// TwinCAT 3 PLC project Untitled1
// ProgramVersion: 3.1.4024.0
// libraries:
//   CmpBitmapPool, * (System)
//   Tc2_EtherCAT, * (Beckhoff Automation GmbH)
//   Tc2_MC2, * (Beckhoff Automation GmbH)
//   Tc2_ModbusSrv, * (Beckhoff Automation GmbH)
//   Tc2_Standard, * (Beckhoff Automation GmbH)
//   Tc2_SUPS, * (Beckhoff Automation GmbH)
//   Tc2_System, * (Beckhoff Automation GmbH)
//   Tc2_Utilities, * (Beckhoff Automation GmbH)
//   Tc3_Module, * (Beckhoff Automation GmbH)
//   Tc3_PackML_V2, * (Beckhoff Automation GmbH)
//   Util, * (System)
//   VisuDialogs, * (System)
// project tree:
//   02DUTs/ E_PMLUserUnitMode.TcDUT, E_UnitName.TcDUT, ST_ChangeIntoProduction.TcDUT (not stored), ST_UnitInfo.TcDUT (not stored)
//   Ads/ BarcodeVerificationResult.TcDUT (not stored), CurrentAirPressureState.TcDUT, DigitalInputStatus.TcDUT (not stored), DigitalOutputStatus.TcDUT (not stored), EStopStatus.TcDUT (not stored), E_SAFETYDOOR.TcDUT, E_SafetyStates.TcDUT (not stored), FB_AirPressure_Subsystem.TcPOU, FB_Application.TcPOU, FB_Light_tower_module.TcPOU (not stored), FB_Safety_module.TcPOU, FB_Tote_Subsystem.TcPOU, MachineControlCommand.TcDUT (not stored), MachineStatus.TcDUT (not stored), SafetyDoorStatus.TcDUT (not stored), SafetyStatus.TcDUT (not stored), StationMode.TcDUT (not stored), ST_LightTower.TcDUT (not stored)
//   GVLs/ GVL.TcGVL, GVL_IOLink.TcGVL (not stored), G_HMI.TcGVL, G_IO.TcGVL, ST_IO_16.TcDUT (not stored), ST_SafetyIO.TcDUT (not stored)
//   / EtherCAT_Task.TcTTO (not stored), GlobalTextList.TcGTLO, MianTask.TcTTO (not stored), VisualizationManager.TcVMO (not stored), VISU_TASK.TcTTO (not stored)
//   Mian/axis/ AxisHMI_Ex.TcVIS (not stored), E_HomingSteps.TcDUT (not stored), FB_MotionAxis_MC.TcPOU (not stored), MC_HomeAxis.TcPOU (not stored), ST_MotionAxis_MC.TcDUT
//   Mian/DUTs/ Buffer_roller.TcDUT (not stored), E_Condition.TcDUT (not stored), E_LoadingStates.TcDUT, E_SampleStates.TcDUT (not stored), E_RollerStates.TcDUT (not stored), E_topic_sample.TcDUT (not stored), E_Transfer.TcDUT (not stored), E_WorkingStates.TcDUT, FB_DigitalInput.TcPOU (not stored), FB_GPWM.TcPOU (not stored), Roller.TcDUT (not stored), ServerityLevelType.TcDUT (not stored), ST_control_pannel.TcDUT (not stored), ST_EVENT.TcDUT (not stored), ST_safetyDoor.TcDUT (not stored), ToteStatus.TcDUT, Valve.TcDUT (not stored)
//   Mian/ FB_mcp.TcPOU (not stored), FB_Generic.TcPOU, FB_Machine.TcPOU, FB_Sample.TcPOU, FB_Visu.TcPOU, I_Common.TcIO, MAIN.TcPOU
//   Mian/statemachine/ Prepare_Date_Time.TcPOU (not stored)
//   PubSub/ E_Topics.TcDUT, I_PubSubService.TcIO, I_SubCallback.TcIO (not stored), KeyAndValue.TcDUT (not stored), PubSubData.TcDUT (not stored), PubSubService.TcPOU, SubscriberCell.TcDUT
//   VISUs/ ImagePool.TcIPO (not stored), visu_main.TcVIS
//   VISUs/Templates/ VIS_TemplateCommand.TcVIS, VIS_TemplateKeys.TcVIS, VIS_TemplateMachine.TcVIS, VIS_TemplatePMLStateModel.TcVIS (not stored), VIS_TemplateToProduction.TcVIS (not stored)
//   VISUs/VISUs/ Menu.TcVIS, visu_sample.TcVIS (not stored), visu_manual.TcVIS, visu_operation.TcVIS, v_alarm.TcVIS
// real-time tasks:
//   TASK PlcTask: cycle T#4ms, priority 20, ADS port 350
//   TASK EtherCAT_Task: cycle T#2ms, priority 2, ADS port 351
//   TASK VISU_TASK: cycle T#100000us, priority 30, ADS port 352
// motion (NC):
//   TASK NC-Task 1 SAF: cycle T#2ms, priority 4, ADS port 501
//   TASK NC-Task 1 SVB: cycle T#10ms, priority 8, ADS port 511
//   AXIS buffer_stopper (id 1)
//     PositionAreaControl: Enable=false
//     OtherSettings: AllowMotionCmdToSlave=true
//     encoder EncType=19
//       EncPara: ScaleFactorNumerator=36, ScaleFactorDenominator=8388608, MaxCount=#xffffffff, ReferenceSystem=1
//         Inc: RefSoftSyncMask=#x00800000
//     drive DrvType=16
//       DrvPara: MaxCount=#xffffffff, DriveControlDWord=#x00000100
//         Analog: TorqueSetpointScale=10, ScaleFactorActTorque=0.1
//         TimeComp: TaskDelayCycles=1
//     controller CtrType=1
//       CtrPara: PriorControlFactor=1
//         PosDiffControl: Enable=false
//         Observer: BandWidth=20
//   AXIS lift_motor (id 3)
//     PositionAreaControl: Enable=false
//     OtherSettings: AllowMotionCmdToSlave=true
//     encoder EncType=19
//       EncPara: ScaleFactorNumerator=3.97364299e-07, MaxCount=#xffffffff, ReferenceSystem=1
//     drive DrvType=16
//       DrvPara: MaxCount=#xffffffff, DriveControlDWord=#x00000100
//         Analog: TorqueSetpointScale=10, ScaleFactorActTorque=0.1
//         TimeComp: TaskDelayCycles=1
//     controller CtrType=1
//       CtrPara: PriorControlFactor=1
//         PosDiffControl: Enable=false
//         Observer: BandWidth=20
//   AXIS working_lift_motor (id 4)
//     PositionAreaControl: Enable=false
//     OtherSettings: AllowMotionCmdToSlave=true
//     encoder EncType=19
//       EncPara: ScaleFactorNumerator=5.96046448e-07, Inverse=true, MaxCount=#xffffffff, ReferenceSystem=1
//     drive DrvType=16
//       DrvPara: Inverse=true, MaxCount=#xffffffff, DriveControlDWord=#x00000100
//         Analog: TorqueSetpointScale=10, ScaleFactorActTorque=0.1
//         TimeComp: TaskDelayCycles=1
//     controller CtrType=1
//       CtrPara: PriorControlFactor=1
//         PosDiffControl: Enable=false
//         Observer: BandWidth=20
//   AXIS working_open_bag (id 5)
//     General: UnitName=°
//     Dynamic: Acceleration=75, Deceleration=75, Jerk=112.5
//     Velo: Maximum=300
//     PositionAreaControl: Enable=false
//     OtherSettings: AllowMotionCmdToSlave=true
//     encoder EncType=19
//       EncPara: ScaleFactorNumerator=36, ScaleFactorDenominator=8388608, MaxCount=#xffffffff, ReferenceSystem=1
//         Inc: RefSoftSyncMask=#x00800000
//     drive DrvType=16
//       DrvPara: MaxCount=#xffffffff, DriveControlDWord=#x00000100
//         Analog: TorqueSetpointScale=10, ScaleFactorActTorque=0.1
//         TimeComp: TaskDelayCycles=1
//     controller CtrType=1
//       CtrPara: PriorControlFactor=1
//         PosDiffControl: Enable=false
//         Observer: BandWidth=20

// ---- 02DUTs/E_PMLUserUnitMode.TcDUT
//Enumeration for User Modes
TYPE E_PMLUserUnitMode : (
	ePMLUnitMode_Service		:=  4,
	ePMLUnitMode_Usermode2		:=  5,
	ePMLUnitMode_Usermode3		:=  6,
	ePMLUnitMode_Usermode4		:=  7,
	ePMLUnitMode_Usermode5 		:=  8,
	ePMLUnitMode_Usermode6 		:=  9,
	ePMLUnitMode_Usermode7 		:=  10
) DINT;
END_TYPE

// ---- 02DUTs/E_UnitName.TcDUT
//Enumeration for Machineunits
TYPE E_UnitName :
(
	eMachine		:= 1,
	eSample			:= 2
				
)DINT;
END_TYPE

// ---- Ads/CurrentAirPressureState.TcDUT
{attribute 'qualified_only'}
{attribute 'strict'}
TYPE CurrentAirPressureState :
(
	UNKNOWN := 0,
	ERROR	:= 1,
	WARNING := 2,          
    HEALTH  := 3,      
    OVERTOP := 4       

);
END_TYPE

// ---- Ads/E_SAFETYDOOR.TcDUT
{attribute 'qualified_only'}
{attribute 'strict'}
TYPE E_SAFETYDOOR :
(
	IDLE := 0,
	SAFETY,
	UNLOCKING,
	UNLOCKED,
	LOCKED,
	WAIT_LOCKED,
	WAIT_UNLOCKED,
	REQUEST_LOCK,
	WAIT_ROBOT
);
END_TYPE

// ---- Mian/axis/ST_MotionAxis_MC.TcDUT
TYPE ST_MotionAxis_MC :
STRUCT
	rVelocity						: 	LREAL   						;
	rVelocity2						: 	LREAL   						;
	rMaxVelocity					:	LREAL							;	
	rAcceleration					:	LREAL							;
	rMaxAcceleration				:	LREAL							;
	rDeceleration					:	LREAL   						;
	rMaxDeceleration				:	LREAL							;
	rJerk							:	LREAL							;
	rMaxJerk						:	LREAL							;
	rPosition						:	LREAL							;
	rSetPosDistance					:	LREAL							;
	rSetPos							: 	LREAL							;	
	rDistance						:   LREAL							;
	rDistance2						:   LREAL							;	
	
	rActualPosSet					:	LREAL							;//ADD BY EVAN 
	rVelocitySet					: 	LREAL   						;//ADD BY EVAN 	
	xHoming							:	BOOL							;//ADD BY EVAN 
	
	rMaxDistance					:	LREAL							;
	bLimit							:   BOOL							;
	bNegLim							:   BOOL							;
	bPosLim							:	BOOL							;
	bNegSen							:   BOOL							;
	bPosSen							:	BOOL							;
	bPositionSensor					:	BOOL							;
	rHomePos						:	LREAL							;
	rActualPos						:	LREAL							;
	PosDiff							:	LREAL							;
	rActualCurr						:	LREAL							;
	axisDirection					:	MC_Direction					;
	
	rVeloPers						: 	LREAL							;
	rAccPers						: 	LREAL							;   
	rDecPers						: 	LREAL							;                                             					
	SetHomePos						: 	LREAL							;
	HomeVelo						: 	LREAL							;
	PosDiffTarget					: 	LREAL							;
	rFirstpos						: 	LREAL							;
	iAxisID							:	INT								;
	xhsHomingStart					: 	BOOL							;
	xHomingDone						: 	BOOL							;
	xForceControlStart				: 	BOOL							;
	xFoceControlDone				:	BOOL							;	
	xMoveABSDone					: 	BOOL							;
	xMoveRelDone					:	BOOL							;
	bInCouple						:	BOOL							;//Flag Axis is coupled 
    xMuteAxisErrorMessages			:	BOOL							;                                         					
	//Visible/Hide HMI interfaces                   					
	bHomeButtonShow					:	BOOL							; 
	bNegSensorShow					:	BOOL							; 
	bPosSensorShow					:	BOOL							;
	bBacklashShow					:	BOOL							;
	bUnitDegShow					:	BOOL							;
    bJerkShow						:	BOOL							; 
	bStopButtonShow					:	BOOL							; 
	   
	
	bMoveAbsHMI						:	BOOL;
	rVelocityHMI 					: 	LREAL;
	rActualPosHMI					:	LREAL							;//ADD BY EVAN
	bMChomingEnable					:	BOOL							;                                         				
	// backlash compensation                        	
	rBacklashvalue					:	LREAL							;
	xbacklashEnable					:	BOOL							;                        		                					
	bdirFW							:	BOOL							;// on hard stop homing , define the direction of rotation
	
	ModOp					 		: 	SINT							;// Axis operation mode (8 )

//	==============================	Beckhoff Tc2_MC2 library(motion)	==================================
	mcPower 						: 	MC_Power					    ;(*	Axis power, enable/disable																			*)
	mcAxisStates					:	MC_AxisStates					;(*	Driver Feedback, curr motor stage 																	*)
	mcHalt							: 	MC_Halt							;(*	Stops an axis with a defined braking ramp															*)
	mcHome							: 	MC_Home							;(*	Axis homing scenario and execution																	*)
	mcJog							: 	MC_Jog							;(*	Axis Joging BW/FW																					*)	
	mcMoveAbsolute					: 	MC_MoveAbsolute					;(*	Axis GoTo Absolute position																			*)	
	mcMoveRelative					: 	MC_MoveRelative					;(*	Axis GoTo Step by SetPos +/- actual position														*)
	mcMoveVelocity					: 	MC_MoveVelocity					;(*	Axis GoTo with constant velocity														*)
	mcReadStatus					: 	MC_ReadStatus					;(*	Read Axis statuses from driver																		*)
	mcReset							: 	MC_Reset						;(*	Reset Driver																						*)
	mcStop							: 	MC_Stop							;(*	Stop Driver																							*)
	mcReadActualPosition			:	MC_ReadActualPosition			;(*	Read the current axis position																		*)
	mcSetpoint						: 	MC_SetPosition					;(*	Sets the current axis position to a parameterizable value											*)
	mcWriteBoolParameter			: 	MC_WriteBoolParameter			;(*	Write bool param to driver																			*)
	mcReadBoolParameter				:	MC_ReadBoolParameter			;(*	Read bool param from driver																			*)
	mcAxisParameter					:   MC_AxisParameter				;(*	Data type is used in conjunction with function blocks for reading and writing of axis parameters	*)
	CoeWrt							:	FB_EcCoESdoWrite;									
	
//	======================================================================================================	

//
	iSdoWrite	:INT; //6:clear encoder
	sNetID : STRING;
	nSlaveAddr	:UINT;
	nSubIndex	: BYTE;
	nIndex	: WORD;
	
	iCoeWrt	: INT;
	rToqueLimitSet	: LREAL	:= 350;
	rToqueSet	: LREAL;
	rActTorque	AT%I*	: LREAL ;
	xTorqueErr	: BOOL;
	bTouchTorque		: BOOL;
	bTouque_control_enable	: BOOL;
	iAxis	: WORD;
	digitalInputs     AT%I*  : UDINT;//bit16:limit_positive;bit17:limit_negative;bit18:limit_home//inovance
END_STRUCT
END_TYPE

// ---- Mian/DUTs/E_LoadingStates.TcDUT
{attribute 'qualified_only'}
{attribute 'strict'}
TYPE E_LoadingStates :
(
	IDLE := 0,
	INIT,
	CHECK,
	WAIT,
	WAIT_1,
	DETECTION,
	LOADING,
	UNLOADING,
	WAIT_NEXT_READY,
	LIFT_POSITION_LOAD,
	LIFT_POSITION_UNLOAD,
	LIFT_UP,
	ROLLER_LOAD,
	ROLLER_UNLOAD,
	WAIT_LEFT_MUTE_OFF,
	WAIT_RIGHT_MUTE_OFF,
	AGING_STATE_0,
	AGING_STATE_1,
	DONE,
	LOAD_UP_POSITION,
	LOAD_DOWN_POSITION,
	ROLLER_Y_LOAD,
	ERROR
);
END_TYPE

// ---- Mian/DUTs/E_WorkingStates.TcDUT
{attribute 'qualified_only'}
{attribute 'strict'}
TYPE E_WorkingStates ://can't divide into 2 states for load and unload,for sometimes if not unload,then call load,can cause accident
(
	IDLE := 0,
	INIT,
	CHECK,
	WAIT_NEW_TOTE,
	LOADING,
	WAIT_FINISHED,
	TOTE_LOAD,
	TOTE_UNLOAD,
	BAG_OPEN,
	BAG_OPEN_DETECTION,
	BAG_CLOSE_STEP_0,
	BAG_CLOSE_STEP_1,
	BAG_CLOSE,
	TOTE_LIFT_UP,
	TOTE_LIFT_DOWN,
	BAG_OPEN_UP,
	BAG_OPEN_DOWN,
	TOTE_OUT,
	WAIT_1,
	
	WAIT_LOGTECH_OUTBOUND,
	TOTE_STATUS_DETECTION,
	
	
	AGING_STATE_0,
	AGING_STATE_1,

	WAIT,
	
	WAIT_UNLOADING,
	WAIT_SENSOR_ON,
	WAIT_SENSOR_OFF,
	WAIT_MUTE_SENSOR_ON,
	WAIT_MUTE_SENSOR_OFF,
	WAIT_LOAD_SENSOR_ON,
	WAIT_LOAD_SENSOR_OFF,
	WAIT_RECEIVE_TOTE_FINISHED,
	WAIT_TOTE_DETECTION_ON,
	WAIT_TOTE_DETECTION_OFF,
	DONE				:= 100,
	ERROR				:= 200
	
);
END_TYPE

// ---- Mian/DUTs/ToteStatus.TcDUT
{attribute 'qualified_only'}
{attribute 'strict'}
TYPE ToteStatus:
(
	UNKNOWN 		:= 0,
	EMPTY 			:= 1,
	LOADED			:= 2,
    READY			:= 3

);
END_TYPE

// ---- PubSub/E_Topics.TcDUT
TYPE E_Topics :
(
	UNKNOWN 				:= 0, 
	SAMPLE_SUBSCRRIBE_1		:= 1, 
	SAMPLE_SUBSCRRIBE_2		:= 2, 
	SAMPLE_SUBSCRRIBE_3		:= 3,
	NUMBER_OF_TOPICS
);
END_TYPE

// ---- PubSub/SubscriberCell.TcDUT
TYPE SubscriberCell :
STRUCT
	occupied : BOOL;
	subscriber : I_SubCallback;
END_STRUCT
END_TYPE

// ---- GVLs/GVL.TcGVL
{attribute 'qualified_only'}
VAR_GLOBAL

	fb_mcp		: FB_mcp;
	
	status	: MachineStatus := MachineStatus.STOPPED;
	
	iAng_air AT%I* :INT;
	aiFlow AT%I* :INT;


	PackTags					: ST_PackMLv30;					//PackTags

	nVisuProductCommand			: DINT;							//Products to produce

	bButtonProductionReq		: BOOL;							//TRUE when a mode change to PRODUCTION is requested
	stChangeIntoProduction		: ST_ChangeIntoProduction;		//Result of command box "Change to Production requested"

	aUnitInfo					: ARRAY [1..12] OF ST_UnitInfo;	//Array includes the states and modes of machineunits	
	aCaption					: ARRAY [1..12] OF STRING := ['F1','F2','F3','F4','F5','F6','F7','F8','F9','F10','F11','F12'];
	aKeyPressed					: ARRAY [1..12] OF BOOL;		
	
	alarm_empty		: ST_Alarm;
	alarm			: ST_Alarm;
	str				: STRING;
	pml_adminAlarm	: PML_AdminAlarm;		
	

	fb_sample	: FB_Sample;
	
	PubSubService	: PubSubService;
END_VAR
VAR_GLOBAL CONSTANT
	iAlarm_max	:INT	:= 19;
	rAir_setting	: REAL	:=0.4;
	MAX_PUB_SUB_DATA	: INT:=19;
END_VAR

// ---- GVLs/G_HMI.TcGVL
{attribute 'qualified_only'}
VAR_GLOBAL
	iMainFrame 		: INT;
	iPML_mainFrame	: INT;

	bInit			: BOOL;
	bAging_test		: BOOL	:= FALSE;
	
	sLoginnedUser	: STRING;
END_VAR

// ---- GVLs/G_IO.TcGVL
{attribute 'global_init_slot' := '40600'}
VAR_GLOBAL CONSTANT
	{attribute 'global_init_slot'}
	DiMouduleMAX 			:	INT	:=	10;
	{attribute 'global_init_slot'}
	DOMODULEMAX 			:	INT	:=	10;
	{attribute 'global_init_slot'}
	SiMouduleMAX 			:	INT	:=	10;
	{attribute 'global_init_slot'}
	SoMODULEMAX 			:	INT	:=	10;	
END_VAR

VAR_GLOBAL
	arDI	AT%I*		: ARRAY[0..DiMouduleMAX ] OF ST_IO_16;		//  links to Digital input  Modules 
	arDO	AT%Q*		: ARRAY[0..DOMODULEMAX ] OF ST_IO_16;		//  links to Digital output Modules	
	arSI	AT%I*		: ARRAY[0..SiMouduleMAX ] OF ST_SafetyIO;	//  links to safety input  Modules
	arSO	AT%I*		: ARRAY[0..SOMODULEMAX ] OF ST_SafetyIO;	//  links to safety output  Modules
END_VAR

// ---- Mian/I_Common.TcIO
INTERFACE I_Common

METHOD GenerateErrorMsg : STRING
VAR_INPUT
	errorType	: STRING;
	strState	: STRING;
	iState		: INT;
	errorMsg	: STRING;
END_VAR
END_METHOD

METHOD GenerateLogMsg : STRING
VAR_INPUT
END_VAR
END_METHOD

METHOD M_Init : BOOL
VAR_INPUT
END_VAR
END_METHOD

METHOD ParseStateToString : STRING
VAR_INPUT
END_VAR
END_METHOD

END_INTERFACE

// ---- PubSub/I_PubSubService.TcIO
(*
Description:
An interface to form the contract for a basic Publisher/Subscriber service.
explaination for each method is located at the method's place.
*)
INTERFACE I_PubSubService

(*
Description:
Through this method you can publish data to a certain topic domain

Params: topic - the type of topic you wish to publish data to.
Params: data - the data you wish to send to said topic.
*)
METHOD Publish
VAR_INPUT
	topic : E_Topics;
	data  : PubSubData;
END_VAR
END_METHOD

(*
Description:
Through this method you can subcribe to a topic and be notified via the I_SubCallback interface.

Params: topic - the type of topic you wish to subscribe to
Params: subCallback - is a reference to subscribe who needs to implement the O_SubCallback interface.
Return: INT - this is an ID you need to keep in order to be able to use the Unsubscribe method.
		ID > 0 is a valid ID, ID = -1 meaning the you've failed to subscribe.
*)
METHOD Subscribe : INT
VAR_INPUT
	topic : E_Topics;
	subCallback :  I_SubCallback;
END_VAR
END_METHOD

(*
Description:
Through this method you can unsubcribe to a topic you've already subscribed beforehand.

Params: topic - the type of topic you wish to unsubscribe to
Params: subscriberID - the ID you've received from the subscribe method.
*)
METHOD Unsubscribe
VAR_INPUT
	topic : E_Topics;
	subscriberID : INT;
END_VAR
END_METHOD

END_INTERFACE

// ---- Mian/FB_Sample.TcPOU
FUNCTION_BLOCK FB_Sample EXTENDS FB_Generic
VAR_INPUT
END_VAR
VAR_OUTPUT
END_VAR
VAR
	lamp			: BOOL;	
	eStates			: E_SampleStates := E_SampleStates.IDLE;;
	eStateTemp		: E_SampleStates := E_SampleStates.IDLE;
	iStateTemp		: INT;	
END_VAR

SUPER^();
IF NOT subscribed THEN
	GVL.PubSubService.Subscribe(E_Topics.SAMPLE_SUBSCRRIBE_1,THIS^);
	GVL.PubSubService.Subscribe(E_Topics.SAMPLE_SUBSCRRIBE_2,THIS^);
	GVL.PubSubService.Subscribe(E_Topics.SAMPLE_SUBSCRRIBE_3,THIS^);
END_IF
subscribed	:= TRUE;


sComponent_name		:= 'fb_sample';
iComponetID			:= 99;
strState	:= ParseStateToString();
infoLevel	:= ServerityLevelType.WARNING;

(*
Description: 
the callback that will be invoked when there is a publish for what the subscriber was subscribed to.
*)
METHOD Callback
VAR_INPUT
	data : PubSubData;
END_VAR
CASE data.Topic OF
	E_Topics.SAMPLE_SUBSCRRIBE_1:
		ADSLOGSTR(msgCtrlMask:= ADSLOG_MSGTYPE_LOG,msgFmtStr:='get data from publish 1',strArg:='');
	E_Topics.SAMPLE_SUBSCRRIBE_2:
		ADSLOGSTR(msgCtrlMask:= ADSLOG_MSGTYPE_LOG,msgFmtStr:='get data from publish 2',strArg:='');
	E_Topics.SAMPLE_SUBSCRRIBE_3:
		ADSLOGSTR(msgCtrlMask:= ADSLOG_MSGTYPE_LOG,msgFmtStr:='get data from publish 3',strArg:='');		
END_CASE
END_METHOD

{attribute 'object_name' := 'M_Aborting'}
METHOD M_Aborting
CASE fbUnitModeManager.eModeStatus OF	
	ePMLProtUnitMode_Production, ePMLProtUnitMode_Manual:		
		lamp	:= FALSE;		
		M_StateComplete();
			
	ePMLProtUnitMode_Maintenance, ePMLUnitMode_Service:
		
		M_StateComplete();
END_CASE
END_METHOD

METHOD M_agingTest : BOOL
VAR_INPUT
	
END_VAR
END_METHOD

{attribute 'object_name' := 'M_Completing'}
METHOD M_Completing
CASE fbUnitModeManager.eModeStatus OF
	ePMLProtUnitMode_Production:
		;
END_CASE
END_METHOD

{attribute 'object_name' := 'M_Execute'}
METHOD M_Execute

CASE fbUnitModeManager.eModeStatus OF
	ePMLProtUnitMode_Production:		//Mode Production
		//////////////////////////////////////////////////////////timeout//////////////////////////////////////////	
		iStateTemp	:= eStateTemp;
		ton_timeout();
		IF eStateTemp=eStates THEN
			ton_timeout.IN	:=TRUE;
		ELSE
			ton_timeout.IN	:=FALSE;
			eStateTemp	:= eStates;	
			M_Log(eLogType:=ServerityLevelType.INFO,sTextLog:='');
			IF ton_timeout.Q THEN
				RETURN;
			END_IF
		END_IF
		IF ton_timeout.Q THEN	
			ton_timeout.IN	:=FALSE;
			CASE eStates OF	
				E_SampleStates.ERROR:	
					alarm_temp.Message	:= GenerateErrorMsg(errorType:='M',iState := iStateTemp,errorMsg:='in error state.');
				ELSE
				alarm_temp.Message	:= GenerateErrorMsg(errorType:='M',iState := iStateTemp,errorMsg:='time out');
			END_CASE
			
//			CASE eStates OF		
//				E_SampleStates.IDLE:						
//					;
//				E_SampleStates.INIT:
//					;
//				E_SampleStates.WAIT_ON:
//					;
//				E_SampleStates.WAIT_OFF:
//					;			
//				E_SampleStates.ERROR:	
//					alarm_temp.Message	:= 'Sample in error state';
//				ELSE
//					alarm_temp.Message	:= 'UNKNOWN STATES in Sample module';
//			END_CASE
			IF eStates<>E_SampleStates.IDLE AND eStates<>E_SampleStates.WAIT_ON AND eStates<>E_SampleStates.WAIT_OFF THEN
				GVL.pml_adminAlarm.M_SetAlarm(stAdmin:=GVL.PackTags.Admin,stAlarm:=alarm_temp);
			END_IF
		END_IF
		
		CASE eStates OF 
				E_SampleStates.IDLE:
					ton_timeout.PT	:= T#1MS;						
					eStates	:= E_SampleStates.INIT;				
				E_SampleStates.INIT:
					ton_timeout.PT	:= T#1S;
					eStates	:= E_SampleStates.WAIT_ON; 
				E_SampleStates.DETECTION:
					ton_timeout.PT	:= T#3S;
				E_SampleStates.WAIT:
					ton_timeout.PT	:= T#200MS;					
				E_SampleStates.WAIT_ON:
					lamp	:= TRUE;
					IF ton_timeout.Q THEN
						eStates	:= E_SampleStates.WAIT_OFF;
					END_IF
				E_SampleStates.WAIT_OFF:
					lamp	:= FALSE;
					IF ton_timeout.Q THEN
						eStates	:= E_SampleStates.IDLE;
					END_IF
				E_SampleStates.ERROR:
					;
			END_CASE
		
		
	ePMLProtUnitMode_Maintenance, ePMLUnitMode_Service:		
		//
		
	ePMLProtUnitMode_Manual:		//Manaul

END_CASE
END_METHOD

{attribute 'object_name' := 'M_Holding'}
METHOD M_Holding
CASE fbUnitModeManager.eModeStatus OF
	ePMLProtUnitMode_Production:		//Mode Production
		//Finisch the actual seperationstep	
		

	ePMLProtUnitMode_Maintenance:
		M_StateComplete();
END_CASE
END_METHOD

{attribute 'object_name' := 'M_Idle'}
METHOD M_Idle
IF G_HMI.bAging_test THEN
	//M_agingTest();
END_IF
END_METHOD

METHOD M_mapping : BOOL
VAR_INPUT
END_VAR
END_METHOD

METHOD M_Reset
VAR_INPUT
END_VAR
//Take away all commands
IF GVL.stChangeIntoProduction.bYesReset THEN
;
END_IF
END_METHOD

{attribute 'object_name' := 'M_Resetting'}
METHOD M_Resetting
CASE fbUnitModeManager.eModeStatus OF
	ePMLProtUnitMode_Production:		//Production, Mantainance, Manual
		lamp	:= FALSE;
		eStates :=E_SampleStates.IDLE;
		M_StateComplete();
	
	ePMLProtUnitMode_Maintenance, ePMLProtUnitMode_Manual, ePMLUnitMode_Service:
		M_StateComplete();
END_CASE
END_METHOD

{attribute 'object_name' := 'M_Starting'}
METHOD M_Starting
CASE fbUnitModeManager.eModeStatus OF
	ePMLProtUnitMode_Production:		//Production, Mantainance, Manual
		
		M_StateComplete();
	ePMLProtUnitMode_Maintenance, ePMLProtUnitMode_Manual, ePMLUnitMode_Service:
		M_StateComplete();
END_CASE
END_METHOD

{attribute 'object_name' := 'M_Stopping'}
METHOD M_Stopping
CASE fbUnitModeManager.eModeStatus OF
	ePMLProtUnitMode_Production, ePMLProtUnitMode_Manual:
				//////////////////////////////////////////////////////////timeout//////////////////////////////////////////	
		iStateTemp	:= eStateTemp;
		ton_timeout();
		IF eStateTemp=eStates THEN
			ton_timeout.IN	:=TRUE;
		ELSE
			ton_timeout.IN	:=FALSE;
			eStateTemp	:= eStates;	
		END_IF
		IF ton_timeout.Q THEN	
			ton_timeout.IN	:=FALSE;
			CASE eStates OF		
				E_SampleStates.IDLE:						
					;
				E_SampleStates.INIT:
					;
				E_SampleStates.WAIT_ON:
					;
				E_SampleStates.WAIT_OFF:
					;			
				E_SampleStates.ERROR:	
					alarm_temp.Message	:= 'Sample in error state';
				ELSE
					alarm_temp.Message	:= 'UNKNOWN STATES in Sample module';
			END_CASE
			IF eStates<>E_SampleStates.IDLE AND eStates<>E_SampleStates.WAIT_ON AND eStates<>E_SampleStates.WAIT_OFF THEN
				GVL.pml_adminAlarm.M_SetAlarm(stAdmin:=GVL.PackTags.Admin,stAlarm:=alarm_temp);
			END_IF
		END_IF
		
		CASE eStates OF 
				E_SampleStates.IDLE:						
					eStates	:= E_SampleStates.INIT;				
				E_SampleStates.INIT:
					ton_timeout.PT	:= T#1S;
					eStates	:= E_SampleStates.WAIT_ON; 
				E_SampleStates.WAIT_ON:
					lamp	:= TRUE;
					IF ton_timeout.Q THEN
						eStates	:= E_SampleStates.WAIT_OFF;
					END_IF
				E_SampleStates.WAIT_OFF:
					lamp	:= FALSE;
					IF ton_timeout.Q THEN
						eStates	:= E_SampleStates.IDLE;
						M_StateComplete();	
					END_IF
				E_SampleStates.ERROR:
					;
			END_CASE			
	ePMLProtUnitMode_Maintenance, ePMLUnitMode_Service:
		M_StateComplete();	
			//not defined
END_CASE
END_METHOD

{attribute 'object_name' := 'M_Undefined'}
METHOD M_Undefined

bUndefinedDone					:= TRUE;
END_METHOD

METHOD ParseStateToString : STRING
VAR_INPUT
END_VAR
CASE THIS^.eStates OF
	E_SampleStates.IDLE:
		ParseStateToString	:='IDLE';
	E_SampleStates.INIT:
		ParseStateToString	:='INIT';
	E_SampleStates.CHECK:
		ParseStateToString	:='CHECK';
	E_SampleStates.DETECTION:	
		ParseStateToString	:='DETECTION';
	E_SampleStates.LAMP_ON:
		ParseStateToString	:='LAMP_ON';
	E_SampleStates.LAMP_OFF:
		ParseStateToString	:='LAMP_OFF';
	E_SampleStates.WAIT:
		ParseStateToString	:='WAIT';
	E_SampleStates.WAIT_ON:
		ParseStateToString	:='WAIT_ON';
	E_SampleStates.WAIT_OFF:
		ParseStateToString	:='WAIT_OFF';
	E_SampleStates.DONE:	
		ParseStateToString	:='DONE';
	E_SampleStates.ERROR:
		ParseStateToString	:='ERROR';
	ELSE
		ParseStateToString	:='UNKNOW STATE';
END_CASE
END_METHOD

END_FUNCTION_BLOCK

// ---- Mian/FB_Generic.TcPOU
//the functionblock FB_Generick is transmitted to every machineunit
FUNCTION_BLOCK FB_Generic IMPLEMENTS ITF_UnitState,I_SubCallback,I_Common
VAR_INPUT
	eModeCommand			: DINT;									//Mode from superior Unit
	eCommand				: E_PMLCommand := ePMLCommand_Abort;	//Command for a new state from superior unit
END_VAR
VAR_OUTPUT
	eMode					: DINT;									//Actual mode of the Unit
	eState					: E_PMLState (*:= ePMLState_Aborted*) ;	//Actual state of the Unit
	
	bUndefinedDone			: BOOL;									//When the SPS is started, the first state is Undefiend. bUndefined is TRUE, when the method Undefined has succesful finished
	bInvalidModeCommandOut	: BOOL;
	bChangeIntoProduction	: BOOL;
END_VAR
VAR
	fbUnitModeManager		: PML_UnitModeManager;					//The PML_UnitModeManager manage the Modechanges
	fbStateMachine 			: PML_StateMachine;						//The PML_StateMachine mangae the Statechanges
	
	nStateModeChange		: INT	:= 0;							//Variable to handle the modechange
	nLastState				: E_PMLState;							//Variable to store last state
	
	packTags				: ST_PackMLv30;
	i	: INT;
	
	ton_timeout			: TON;
	
	rTrig_electricalError	:ARRAY[0..10] OF R_TRIG;
	alarm_temp		: ST_Alarm;
	subscribed	: BOOL	:= FALSE;
	subData		: PubSubData;
	
	strState	: STRING;
	sComponent_name			: STRING;
	iComponetID				: INT;	
	infoLevel	: ServerityLevelType;//should be set to high level after debug
END_VAR

M_mapping();
CASE nStateModeChange OF
0:
	//Waiting for user request
	bChangeIntoProduction:= FALSE;
	IF  GVL.bButtonProductionReq AND (GVL.PackTags.Command.UnitMode = ePMLProtUnitMode_Production) AND (GVL.PackTags.Status.UnitModeCurrent = ePMLProtUnitMode_Invalid) THEN
			nStateModeChange	:= 1;
	ELSIF  GVL.PackTags.Command.UnitModeChangeRequest AND (GVL.PackTags.Command.UnitMode <> ePMLProtUnitMode_Production) THEN
			nStateModeChange	:= 1;
	ELSIF  GVL.bButtonProductionReq AND (GVL.PackTags.Command.UnitMode = ePMLProtUnitMode_Production) AND (GVL.PackTags.Status.UnitModeCurrent <> ePMLProtUnitMode_Production) THEN
			nStateModeChange	:= 3;
	END_IF
1:
	//Starting UnitModeManager 
	fbUnitModeManager.bExecute				:= TRUE;
	fbUnitModeManager.eModeCommand			:= eModeCommand;
	GVL.PackTags.Status.UnitModeChangeInProcess	:= TRUE;

	IF fbUnitModeManager.bDone THEN
		fbUnitModeManager.bExecute	:= FALSE;
		bInvalidModeCommandOut		:= FALSE;
		nStateModeChange			:= 0;
		bChangeIntoProduction		:= FALSE;
		GVL.PackTags.Status.UnitModeChangeInProcess	:= FALSE;
	ELSIF fbUnitModeManager.bError THEN
		bInvalidModeCommandOut		:= TRUE;
		fbUnitModeManager.bExecute	:= FALSE;
		nLastState					:= GVL.PackTags.Status.StateCurrent;
		nLastState					:= GVL.PackTags.Status.StateCurrent;
		nStateModeChange			:= 2;
		bChangeIntoProduction		:= FALSE;
		GVL.PackTags.Status.UnitModeChangeInProcess	:= FALSE;
	END_IF
2:
	//ErrorHanddling
	IF  GVL.PackTags.Command.UnitModeChangeRequest THEN
		nStateModeChange:=0;
		bInvalidModeCommandOut		:= FALSE;
	ELSIF nLastState<> GVL.PackTags.Status.StateCurrent THEN
		bInvalidModeCommandOut		:= FALSE;
	END_IF
	
3:
	//state to check, if command 'Porduction' is valid
	IF (GVL.PackTags.Status.StateCurrent = ePMLState_Aborted OR GVL.PackTags.Status.StateCurrent = ePMLState_Stopped OR GVL.PackTags.Status.StateCurrent = ePMLState_Idle) THEN
		bChangeIntoProduction		:= TRUE;
		IF  GVL.stChangeIntoProduction.bYes OR GVL.stChangeIntoProduction.bYesReset THEN
			nStateModeChange			:= 1;		
		ELSIF GVL.stChangeIntoProduction.bNo THEN
			nStateModeChange			:= 0;
		END_IF
	ELSE
		nStateModeChange:= 2;
		bInvalidModeCommandOut		:= TRUE;
		nLastState					:= GVL.PackTags.Status.StateCurrent;
	END_IF
END_CASE


fbUnitModeManager(									
	eState			:= eState,
	eModeStatus		=> eMode,
	bDone			=> ,
	bError			=> ,
	nErrorId		=> );


IF fbUnitModeManager.eModeStatus <>  0 THEN
	//Calling the StateMachine, when there is a valid Mode
	fbStateMachine(
		eMode				:= eMode, 				
		eCommand			:= eCommand,			
		stSubUnitInfoRef	:= ,
		stOptions			:= , 
		eState				=> eState, 				
		bError				=> , 
		nErrorID			=> );
END_IF

//One of the methods is executing  by the actual state
CASE eState OF
	ePMLState_Undefined:
		M_Undefined();
	ePMLState_Clearing:
		M_Clearing();
	ePMLState_Stopped:
		M_Stopped();
	ePMLState_Starting:
		M_Starting();
	ePMLState_Idle:
		M_Idle();
	ePMLState_Suspended:
		M_Suspended();
	ePMLState_Execute:
		M_Execute();
	ePMLState_Stopping:
		M_Stopping();
	ePMLState_Aborting:
		M_Aborting();
	ePMLState_Aborted:
		M_Aborted();
	ePMLState_Holding:
		M_Holding();
	ePMLState_Held:
		M_Held();
	ePMLState_Unholding:
		M_Unholding();
	ePMLState_Suspending:
		M_Suspending();
	ePMLState_Unsuspending:
		M_Unsuspending();
	ePMLState_Resetting:
		M_Resetting();
	ePMLState_Completing:
		M_Completing();
	ePMLState_Complete:
		M_Complete();
END_CASE

(*
Description: 
the callback that will be invoked when there is a publish for what the subscriber was subscribed to.
*)
METHOD Callback
VAR_INPUT
	data : PubSubData;
END_VAR
END_METHOD

(*
GenerateErrorMsg method:generate the error message according to the inputs
generate example:'{M9906} fb_sample DETECTION time out for T#3s.'
errorType:
		'M':mechanical error
		'E':electrical error
		'S':safety error
iState:state of state machine
errorMsg:descirbe the error
sComponent_name:defined in every componet
iComponetID:defined in every componet
strState:parseStateToString() to get the strState in ervery component
sTimeout_setting:defined in every componet
*)
METHOD GenerateErrorMsg : STRING
VAR_INPUT
	errorType	: STRING;
	iState		: INT;
	errorMsg	: STRING;	
END_VAR
VAR
	errorID	: INT;
END_VAR
GenerateErrorMsg	:= '';
GenerateErrorMsg	:= CONCAT('{',errorType);
IF iComponetID<10 THEN
	errorID	:= iComponetID*1000+iState;
ELSE
	errorID	:= iComponetID*100+iState;
END_IF
GenerateErrorMsg	:= CONCAT(GenerateErrorMsg,INT_TO_STRING(errorID));
GenerateErrorMsg	:= CONCAT(GenerateErrorMsg,'} ');
GenerateErrorMsg	:= CONCAT(GenerateErrorMsg,sComponent_name);
GenerateErrorMsg	:= CONCAT(GenerateErrorMsg,' ');
GenerateErrorMsg	:= CONCAT(GenerateErrorMsg,strState);
GenerateErrorMsg	:= CONCAT(GenerateErrorMsg,' ');
GenerateErrorMsg	:= CONCAT(GenerateErrorMsg,errorMsg);
IF errorMsg='time out' THEN
	GenerateErrorMsg	:= CONCAT(GenerateErrorMsg,' ');
	GenerateErrorMsg	:= CONCAT(GenerateErrorMsg,'for ');
	GenerateErrorMsg	:= CONCAT(GenerateErrorMsg,TIME_TO_STRING(ton_timeout.PT));//timeout setting
	GenerateErrorMsg	:= CONCAT(GenerateErrorMsg,'.');
END_IF
END_METHOD

{attribute 'object_name' := 'M_Aborted'}
METHOD M_Aborted
END_METHOD

{attribute 'object_name' := 'M_Aborting'}
METHOD M_Aborting
M_StateComplete();
END_METHOD

METHOD M_CheckError : BOOL
VAR_INPUT
END_VAR

VAR
	Trigger: INT;
END_VAR
M_CheckError	:= FALSE;

FOR i:=1 TO GlobalParameters.MaxAlarms DO
	IF THIS^.PackTags.Admin.Alarm[i].Trigger THEN
		M_CheckError	:= TRUE;
	END_IF
END_FOR
END_METHOD

{attribute 'object_name' := 'M_Clearing'}
METHOD M_Clearing
M_StateComplete();
END_METHOD

{attribute 'object_name' := 'M_Complete'}
METHOD M_Complete
END_METHOD

{attribute 'object_name' := 'M_Completing'}
METHOD M_Completing
M_StateComplete();
END_METHOD

{attribute 'object_name' := 'M_Execute'}
METHOD M_Execute

M_StateComplete();
END_METHOD

{attribute 'object_name' := 'M_Held'}
METHOD M_Held
END_METHOD

{attribute 'object_name' := 'M_Holding'}
METHOD M_Holding
M_StateComplete();
END_METHOD

{attribute 'object_name' := 'M_Idle'}
METHOD M_Idle
END_METHOD

METHOD M_Init : BOOL
VAR_INPUT
END_VAR
END_METHOD

(*
M_Log method :will be show the text in the TwinCAT output window when using the IDE,and also in the windows event logger
the method will filter out the logs who's type is above the info
*)
METHOD M_Log : STRING
VAR_INPUT
	eLogType	: ServerityLevelType;
	sTextLog	: STRING;	
END_VAR
IF eLogType <= infoLevel THEN
	ADSLOGSTR(msgCtrlMask:=Tc2_System.ADSLOG_MSGTYPE_LOG,msgFmtStr:=strState,strArg:='');	
END_IF
END_METHOD

METHOD M_mapping : BOOL
VAR_INPUT
END_VAR
alarm_temp.DateTime	:=GVL.packTags.Admin.PlcDateTime;
END_METHOD

{attribute 'object_name' := 'M_Resetting'}
METHOD M_Resetting
M_StateComplete();
END_METHOD

{attribute 'object_name' := 'M_Starting'}
METHOD M_Starting
M_StateComplete();
END_METHOD

{attribute 'object_name' := 'M_StateComplete'}
METHOD M_StateComplete
//the actual state is completed
fbStateMachine.M_StateComplete();
END_METHOD

{attribute 'object_name' := 'M_Stopped'}
METHOD M_Stopped
END_METHOD

{attribute 'object_name' := 'M_Stopping'}
METHOD M_Stopping
M_StateComplete();
END_METHOD

{attribute 'object_name' := 'M_Suspended'}
METHOD M_Suspended
END_METHOD

{attribute 'object_name' := 'M_Suspending'}
METHOD M_Suspending
VAR_INPUT
END_VAR
M_StateComplete();
END_METHOD

{attribute 'object_name' := 'M_Undefined'}
METHOD M_Undefined
END_METHOD

{attribute 'object_name' := 'M_Unholding'}
METHOD M_Unholding
VAR_INPUT
END_VAR
M_StateComplete();
END_METHOD

{attribute 'object_name' := 'M_Unsuspending'}
METHOD M_Unsuspending
VAR_INPUT
END_VAR
M_StateComplete();
END_METHOD

METHOD ParseStateToString : STRING
VAR_INPUT
END_VAR
END_METHOD

END_FUNCTION_BLOCK

// ---- PubSub/PubSubService.TcPOU
FUNCTION_BLOCK PubSubService IMPLEMENTS I_PubSubService
VAR_INPUT
END_VAR
VAR_OUTPUT
END_VAR

VAR
	TopicsToSubscribers : ARRAY[0..MAX_TOPICS - 1, 0..MAX_SUBSCRIBERS_PER_TOPIC - 1] OF SubscriberCell;
	subscriberCounters : ARRAY [0..MAX_TOPICS - 1] OF INT;
END_VAR

VAR CONSTANT 
	MAX_SUBSCRIBERS_PER_TOPIC : INT := 20;
	{attribute 'analysis' := '-33'}
	MAX_TOPICS : INT := E_Topics.NUMBER_OF_TOPICS;
END_VAR

METHOD Publish
VAR_INPUT
	topic	: E_Topics;
	data	: PubSubData;
END_VAR
VAR
	index : INT;
END_VAR
FOR index := 0 TO MAX_SUBSCRIBERS_PER_TOPIC -1 BY 1 DO
	IF TopicsToSubscribers[topic, index].OCCUPIED = TRUE THEN
		TopicsToSubscribers[topic, index].subscriber.Callback(data);
	END_IF
END_FOR
END_METHOD

METHOD Subscribe : INT
VAR_INPUT
	topic	: E_Topics;
	subCallback	: I_SubCallback;
END_VAR
VAR 
	index : INT;
END_VAR
Subscribe := -1;

IF  subscriberCounters[topic] >= MAX_SUBSCRIBERS_PER_TOPIC THEN
	RETURN;
END_IF

FOR index := 0 TO (MAX_SUBSCRIBERS_PER_TOPIC - 1) BY 1 DO
	IF TopicsToSubscribers[topic, index].occupied = FALSE THEN
		TopicsToSubscribers[topic, index].occupied := TRUE;
		TopicsToSubscribers[topic, index].subscriber := subCallback;
		Subscribe := index;
		subscriberCounters[topic] := subscriberCounters[topic] + 1;
		RETURN;
	END_IF
END_FOR
END_METHOD

METHOD Unsubscribe
VAR_INPUT
	topic : E_Topics;
	subscriberID	: INT;
END_VAR
IF TopicsToSubscribers[topic, subscriberID].occupied = TRUE THEN
	TopicsToSubscribers[topic, subscriberID].occupied := FALSE;
	subscriberCounters[topic] := subscriberCounters[topic] - 1; 	
END_IF
END_METHOD

END_FUNCTION_BLOCK

// ---- Ads/FB_AirPressure_Subsystem.TcPOU
FUNCTION_BLOCK FB_AirPressure_Subsystem
VAR_INPUT
END_VAR
VAR_OUTPUT
END_VAR
VAR
	//current_air_pressure: INT;
	current_air_pressure	: REAL;
	current_air_pressure_state	: CurrentAirPressureState;
	ton1	: TON;
	iCase	 : INT;
	
	
	iFlow	: INT;
	rCurrent_flow	: REAL;
	current_air_flow	: REAL;//unit: L/min
	i1	: INT;
END_VAR
VAR CONSTANT
	air_pressure_threshold_error: REAL:=0.4;//0.4*100 setting in PLC
	air_pressure_threshold_warning: REAL:=0.5;//0.5*100 setting in PLC
	air_pressure_threshold_overtop: REAL:=1;//1*100 setting in PLC
	
	rMin_voltage_flow	: REAL	:= 0.974;
	rMax_voltage_flow	: REAL	:= 5;
	rMaxFlow_L_per_minute		: REAL	:= 2000;
END_VAR

ton1(PT:=T#100MS);

CASE iCase OF
	0:
		ton1.IN	:= TRUE;
		IF ton1.Q THEN
			iCase	:= 1;
		END_IF
	1:
		ton1.IN	:= FALSE;
		//current_air_pressure	:= DINT_TO_INT(GVL.iAng_air*100/16#8000);
		current_air_pressure	:= INT_TO_REAL(GVL.iAng_air)/16#8000;
		IF current_air_pressure<air_pressure_threshold_error THEN
			current_air_pressure_state	:= CurrentAirPressureState.ERROR;
		ELSIF current_air_pressure<air_pressure_threshold_warning THEN
			current_air_pressure_state	:= CurrentAirPressureState.WARNING;
		ELSIF current_air_pressure<air_pressure_threshold_overtop THEN
			current_air_pressure_state	:= CurrentAirPressureState.HEALTH;
		ELSE
			current_air_pressure_state	:= CurrentAirPressureState.OVERTOP;
		END_IF
		
		/////////////////////////////////////////////////

		IF rCurrent_flow>=1 THEN
			current_air_flow	:= rMaxFlow_L_per_minute*(rCurrent_flow-rMin_voltage_flow)/(rMax_voltage_flow-rMin_voltage_flow);
		ELSE
			current_air_flow	:= 0;
		END_IF		
		iCase	:= 0;
	
END_CASE

		rCurrent_flow	:= INT_TO_REAL(GVL.aiFlow*10)/16#8000;

END_FUNCTION_BLOCK

// ---- Ads/FB_Application.TcPOU
FUNCTION_BLOCK FB_Application
VAR_INPUT
END_VAR
VAR_OUTPUT
END_VAR
VAR
	safety : FB_Safety_module;
	tote_subsystem	: FB_Tote_Subsystem;
	light_tower	: FB_Light_tower_module;
	air_pressure_subsystem	: FB_AirPressure_Subsystem;
END_VAR

safety();
light_tower();
tote_subsystem();
air_pressure_subsystem();

GVL.fb_mcp.lightTower := light_tower._lightTower;

END_FUNCTION_BLOCK

// ---- Ads/FB_Safety_module.TcPOU
FUNCTION_BLOCK FB_Safety_module
VAR_INPUT
END_VAR
VAR_OUTPUT
END_VAR
VAR
	SI_0	: UINT;
	SI_1	: UINT;
	GI_0 	: UINT;
	GI_1 	: UINT;
	safety_status	: SafetyStatus	:= SafetyStatus.UNKNOWN;
	
	station_mode	: StationMode;//APP status
	iStationMode	: UINT;
	iState: INT;
	bEstop_detection	: BOOL;	
	
	ton_timeout	: TON;	
	eStates					:	E_SafetyStates	:=	E_SafetyStates.IDLE;
	iStateTemp			: INT;
	errorMessage	: STRING;
	xError	: BOOL;
	eStates_safetyDoor	: E_SAFETYDOOR	:= E_SAFETYDOOR.IDLE;
	bReset_safetyDoor	: BOOL;
	
	
	
	
	
	GPWM	: FB_GPWM;
	GPWM_1s	: FB_GPWM;
	tonSaftyDelay: TON;
	b_EStopRestarting  : BOOL;
	T_EStopRestart : TON;
//////////////////////SAFETY hardware config///////////////	
	mcp_estop	: BOOL;
	mcp_safetyDoor	: BOOL;
	belt_estop	: BOOL;
	lift_estop : BOOL;
	lift_lightCurtain_left	: BOOL;
	lift_lightCurtain_right	: BOOL;
	lift_station_detection	: BOOL;
	
	robot_EES				: BOOL;
	robot_EAS				: BOOL;
	buffer_safety			: BOOL;
	loading_safety			: BOOL;
	working_safety			: BOOL;
//	buffer_safety_24v		: BOOL;
//	buffer_safety_stepmotor	: BOOL;
//	loding_safety_sto		: BOOL;
//	loding_safety_24v		: BOOL;
//	working_safety_sto		: BOOL;
//	working_safety_24v		: BOOL;
	
	pSafety_door	: POINTER TO ST_safetyDoor;
	safety_door_unlock_en		: BOOL;
	bStop_button_unlock		: BOOL;//for not receive cmd from tote_subsystem
	
	ton_wait_robot	: TON;
	
	
	refMachineCmd	: REFERENCE TO E_PMLCommand;
END_VAR

refMachineCmd	REF= MAIN.fbMachine.eCommand;
M_mapping();
M_safetyDoor();
//xError	:=NOT(robot_EES AND buffer_safety AND loading_safety AND working_safety); //if only open the door,machine will just stop,so can control the machine munually
//to do:as below commit and reprogram safety project and test

CASE iState	 OF
	0:
	;

	2:
		IF update_station_mode(2) THEN
			iState	:= 0;
		END_IF	
	3:
		IF M_reset() THEN
			iState	:= 0;
		END_IF
		
END_CASE
//安全Safety报警 确认 复位
tonSaftyDelay(IN:= NOT tonSaftyDelay.Q ,PT:=T#1S);
b_ErrorAck := tonSaftyDelay.Q;



GPWM(i_xEnable:=TRUE,i_udiTime:=25,i_udiCycle:=50);
GPWM_1s(i_xEnable:=TRUE,i_udiTime:=500,i_udiCycle:=1000);

 


 //EDM config
 SPtop_EDM  	  	   := TRUE ;  
 robot_eas_edm  	   := TRUE ;
 light_STO_EDM         := TRUE ;
 PickModule_STO_EDM    := TRUE ;
 Rolller_belt_STO_EDM  := TRUE ;

PROPERTY _stationMode : StationMode
GET
_stationMode	:= station_mode;
END_GET
SET
station_mode	:= _stationMode;
END_SET
END_PROPERTY

METHOD M_mapping : BOOL
VAR_INPUT
END_VAR



mcp_estop					:= SI0_0 AND SI0_1;
mcp_safetyDoor				:= SI0_2 AND SI0_3;
belt_estop					:= SI1_0 AND SI1_1;
lift_lightCurtain_left		:= SI2_0 AND SI2_1;
lift_estop					:= SI2_2 AND SI2_3;
lift_lightCurtain_right		:= SI3_0 AND SI3_1;
lift_station_detection		:= SI3_2 AND SI3_3;
bShield_light_curtain_Left	:= SI4_0;
bShield_light_curtain_Right	:= SI4_1;


robot_EES				:= SO0_0;
robot_EAS				:= SO0_1;
buffer_safety			:= SO1_0;

loading_safety			:= SO2_0;

working_safety			:= SO3_0;

	
	                    
                    
                  
	
IF robot_EES AND robot_EAS THEN 
    safety_status := SafetyStatus.READY ;   //正常
ELSE
	safety_status := SafetyStatus.SAFETY_STOPPED; //急停状态
END_IF

GI_0.0	:= GVL.fb_mcp.st_safety_door.button_reset;
GI_0.1	:= GVL.fb_mcp.st_safety_door.button_unlock;
GI_0.2	:= GVL.fb_mcp.st_safety_door.door_closed;

SI_0.0	:= mcp_estop;
SI_0.1	:= mcp_safetyDoor;
SI_0.2	:= belt_estop;
SI_0.3	:= lift_estop;
SI_0.4	:= lift_station_detection;
END_METHOD

METHOD M_reset : BOOL
VAR_INPUT
	
END_VAR
M_reset	:= FALSE;
xError	:= FALSE;//remove while safety is ready
M_reset	:= TRUE;//remove while safety is ready
RETURN;//remove while safety is ready
//check if all estop
//check if safety door ossd
//check if safety door closed
//lock safety door 
//reset to output safety
//////////////////////////////////////////////////////////timeout//////////////////////////////////////////
ton_timeout();
IF eStates<>E_SafetyStates.IDLE AND eStates<>E_SafetyStates.ERROR  THEN
	IF iStateTemp=eStates THEN
		ton_timeout.IN	:=TRUE;
	ELSE
		ton_timeout.IN	:=FALSE;
		iStateTemp	:= eStates;
	END_IF
ELSE
	ton_timeout.IN	:=FALSE;
END_IF
IF ton_timeout.Q THEN	
	ton_timeout.IN	:=FALSE;
	CASE eStates OF
		E_SafetyStates.DOOR_LOCK:		
			errorMessage	:= CONCAT('door lock error.->safety ',INT_TO_STRING(iStateTemp));
	END_CASE
	IF eStates=E_SafetyStates.DOOR_LOCK AND eStates<>E_SafetyStates.TRIG_RESET THEN
		eStates	:= E_SafetyStates.ERROR;
	END_IF
	
END_IF
CASE eStates OF
	E_SafetyStates.IDLE:
		xError	:= FALSE;
		bReset_safetyDoor	:= FALSE;
		eStates	:= E_SafetyStates.CHECK_ESTOP;
	E_SafetyStates.CHECK_ESTOP:
		IF mcp_estop AND belt_estop AND lift_estop THEN
			eStates	:= E_SafetyStates.CHECK_DOOR_CLOSED;
		ELSE
			eStates	:= E_SafetyStates.ERROR;
		END_IF
	E_SafetyStates.CHECK_DOOR_CLOSED:
		IF GVL.fb_mcp.st_safety_door.door_closed THEN
			eStates	:= E_SafetyStates.DOOR_LOCK;
		ELSE
			eStates	:= E_SafetyStates.ERROR;
		END_IF
	E_SafetyStates.DOOR_LOCK:
		bReset_safetyDoor	:= TRUE;
//		pSafety_door^.door_lock	:= FALSE;
		IF mcp_safetyDoor THEN
			bReset_safetyDoor	:= FALSE;
			eStates	:= E_SafetyStates.TRIG_RESET;
		END_IF		
	E_SafetyStates.TRIG_RESET:
		ton_timeout.PT	:= T#2S;
		b_EStopRestart	:= GPWM.q_xOut;
		IF ton_timeout.Q THEN
			b_EStopRestart	:= FALSE;
			eStates	:= E_SafetyStates.CHECK_SAFETY_OUTPUT;
		END_IF
	E_SafetyStates.CHECK_SAFETY_OUTPUT:	
		IF robot_EES AND robot_EAS AND buffer_safety AND loading_safety AND working_safety THEN
			eStates	:= E_SafetyStates.DONE;
		ELSE
			eStates	:= E_SafetyStates.ERROR;
		END_IF
	E_SafetyStates.DONE:
		M_reset	:= TRUE;
		eStates	:= E_SafetyStates.IDLE;
	E_SafetyStates.ERROR:	
		M_reset	:= TRUE;
		xError	:= TRUE;
		bReset_safetyDoor	:= FALSE;
		eStates	:= E_SafetyStates.IDLE;

	
END_CASE
END_METHOD

METHOD M_safetyDoor : BOOL
VAR_INPUT
	
END_VAR
pSafety_door	:= ADR(GVL.fb_mcp.st_safety_door);
safety_door_unlock_en	:= (safety_status=SafetyStatus.SAFETY_STOPPED OR station_mode = StationMode.STOPPED OR station_mode = StationMode.DISABLED
							OR station_mode = StationMode.FORCE_STOP OR station_mode = StationMode.INTERVENTION OR MAIN.application.tote_subsystem.ton_heart_beat.Q); 
							
ton_wait_robot(PT:=T#500MS);
							
CASE eStates_safetyDoor	 OF
	E_SAFETYDOOR.IDLE:
		IF mcp_safetyDoor THEN
			eStates_safetyDoor	:= E_SAFETYDOOR.LOCKED;
		ELSE
			eStates_safetyDoor	:= E_SAFETYDOOR.UNLOCKED;
		END_IF
	E_SAFETYDOOR.LOCKED:
		pSafety_door^.lamp_reset	:=	FALSE;
		pSafety_door^.lamp_unlock	:= FALSE;
		IF pSafety_door^.button_unlock THEN
			bStop_button_unlock	:= TRUE;
			eStates_safetyDoor	:= E_SAFETYDOOR.WAIT_ROBOT;
		END_IF
	E_SAFETYDOOR.REQUEST_LOCK:
	;
	E_SAFETYDOOR.SAFETY:
	;
	E_SAFETYDOOR.UNLOCKED:
		pSafety_door^.lamp_unlock	:= TRUE;//door unlocked,unlock lamp solid
		IF pSafety_door^.door_closed THEN
			pSafety_door^.lamp_reset	:= GPWM_1s.q_xOut;//door closed,reset lamp blinking
			IF pSafety_door^.button_reset OR bReset_safetyDoor THEN
				bStop_button_unlock	:= FALSE;
				eStates_safetyDoor	:= E_SAFETYDOOR.WAIT_LOCKED;
			END_IF
		ELSE
			pSafety_door^.lamp_reset	:= FALSE;
		END_IF
	E_SAFETYDOOR.WAIT_LOCKED:
		pSafety_door^.door_lock	:= FALSE;
		IF mcp_safetyDoor THEN
			eStates_safetyDoor	:= E_SAFETYDOOR.LOCKED;
	 	END_IF
	E_SAFETYDOOR.WAIT_ROBOT:
			ton_wait_robot.IN := TRUE;
			refMachineCmd	:= ePMLCommand_Stop;
			IF ton_wait_robot.Q THEN
				ton_wait_robot.IN	:= FALSE;
				eStates_safetyDoor	:= E_SAFETYDOOR.UNLOCKING;
			END_IF
	E_SAFETYDOOR.UNLOCKING:
		refMachineCmd	:= ePMLCommand_Stop;
		pSafety_door^.lamp_unlock	:= GPWM_1s.q_xOut;//door opennig,unlock lamp blinking
		IF safety_door_unlock_en THEN
			pSafety_door^.door_lock	:= TRUE;
			IF NOT mcp_safetyDoor THEN
				eStates_safetyDoor	:= E_SAFETYDOOR.UNLOCKED;
			END_IF
		END_IF
	
END_CASE
END_METHOD

{attribute 'TcRpcEnable'}
METHOD update_station_mode  : BOOL
VAR_INPUT
	iMode	: StationMode;
END_VAR
update_station_mode	:= FALSE;
station_mode	:= iMode;
update_station_mode	:= TRUE;
END_METHOD

END_FUNCTION_BLOCK

// ---- Mian/MAIN.TcPOU
// Disclaimer
// 
// This publication contains statements about the suitability of our products for certain areas of application. These statements are based on typical features of our products. The examples shown in this publication are for demonstration purposes only. 
// The information provided herein should not be regarded as specific operation characteristics. It is incumbent on the customer to check and decide whether a product is suitable for use in a particular application. 
// We do not give any warranty that the source code which is made available with this publication is complete or accurate. 
//
// THE SAMPLE CODE CONTAINED IN THIS PUBLICATION IS PROVIDED “AS IS” WITHOUT WARRANTY OF ANY KIND, EITHER EXPRESSED, IMPLIED OR STATUTORY, INCLUDING WITHOUT LIMITATION, ANY WARRANTY WITH RESPECT TO NON-INFRINGEMENT, FREEDOM FROM PROPRIETARY RIGHTS OF THIRD PARTIES OR FITNESS FOR ANY PARTICULAR PURPOSE. 
// This publication may be changed from time to time without prior notice. No liability is assumed for errors and/or omissions. Our products are described in detail in our data sheets and documentations. Product-specific warnings and cautions must be observed. 
// For the latest version of our data sheets and documentations visit our website (www.beckhoff.de). 
//
// © Beckhoff Automation GmbH & Co. KG, 2022
// The reproduction, distribution and utilization of this document as well as the communication of its contents to others without express authorization is prohibited. Offenders will be held liable for the payment of damages. All rights reserved in the event of the grant of a patent, utility model or design.
PROGRAM MAIN
VAR_INPUT
	bExecuteComplete			: BOOL;									//Command Execute Complete, not defined
END_VAR
VAR
	UserModeCofig				: PML_UnitModeConfig;					//User can configure his own Mode
	
	fbMachine					: FB_Machine;							//Instance of FB_Machine
	bMachineStartedUp			: BOOL := FALSE;						//TRUE, when first PLC-Cycle finish

	fbVisu						: FB_Visu;								//Visualization
	
	fbTrigger					: F_TRIG;								//Trigger for resseting Counters

	fbLocalSystemTime			 : FB_LocalSystemTime;					//Get local Systemtime
	
	fbTriggerErrorMainAxis		: R_TRIG;								//Trigger for detecting Error on Mainaxis and write into PackTags
	fbTriggerErrorMetalAxis		: R_TRIG;								//Trigger for detecting Error on Metalaxis and write into PackTags
	fbTriggerErrorPlasticAxis	: R_TRIG;								//Trigger for detecting Error on Plasticaxis and write into PackTags
	
	nStateCommandCheck			: DINT;									//State to handle with statecommands
	
	i	: INT;
	tonDly	: TON;
	
	fb_ups	:FB_S_UPS_CX51x0;
	application	: FB_Application;

	bButton				: BOOL;
	ton_button			: TON;

	refMachine_control_cmd	:REFERENCE TO MachineControlCommand;
	
	
	PackTags					: ST_PackMLv30;	
	rTrig_error	:ARRAY[0..10] OF R_TRIG;
	rTrig_agingTest	:R_TRIG;
	fTrig_agingTest	:F_TRIG;

	
	topicCallbackTest	: E_Topics;
	dataCallbackTest	: PubSubData;
	topic_sample	: E_topic_sample;
	
END_VAR

fb_ups();
GVL.fb_mcp();

application();
refMachine_control_cmd	REF= MAIN.application.tote_subsystem.machine_control_cmd;

tonDly(PT:= T#10MS);
//Configure Usermode 1
A_UnitModeConfig();

//Runs the first PLC-Cycle
IF fbMachine.bUndefinedDone AND NOT bMachineStartedUp THEN
	GVL.PackTags.Command.CntrlCmd	:= ePMLCommand_Abort;
	bMachineStartedUp			:= TRUE;
END_IF


GVL.bButtonProductionReq := GVL.PackTags.Command.UnitMode = ePMLProtUnitMode_Production AND GVL.PackTags.Status.UnitModeCurrent <> GVL.PackTags.Command.UnitMode;


CASE nStateCommandCheck OF	
0:
	tonDly.IN := FALSE;
	GVL.PackTags.Command.CntrlCmd := ePMLCommand_Undefined;
	nStateCommandCheck :=1;
1:	
	tonDly.IN := TRUE;
	IF tonDly.Q THEN
		nStateCommandCheck :=0;
	END_IF
CASE fbMachine.eState OF
			
	ePMLState_Aborted:
		IF (GVL.PackTags.Command.CntrlCmd = ePMLCommand_Clear OR GVL.fb_mcp.st_safety_door.button_reset) THEN
			fbMachine.eCommand	:= ePMLCommand_Clear;
		END_IF
	ePMLState_Complete:		
		IF (GVL.PackTags.Command.CntrlCmd = ePMLCommand_Reset OR refMachine_control_cmd = MachineControlCommand.RESET OR GVL.fb_mcp.st_safety_door.button_reset) THEN
			fbMachine.eCommand	:= ePMLCommand_Reset;
		END_IF
	ePMLState_Idle:
		IF (GVL.PackTags.Command.CntrlCmd = ePMLCommand_Start OR refMachine_control_cmd = MachineControlCommand.START)	
	 	AND (NOT (GVL.PackTags.Command.Parameter[1].Value <= 0) OR NOT (fbMachine.eMode = 1))THEN
			 fbMachine.eCommand	:= ePMLCommand_Start; 
		END_IF
		IF refMachine_control_cmd = MachineControlCommand.RESET THEN
			refMachine_control_cmd	:= MachineControlCommand.DO_NOTHING;
		END_IF
	ePMLState_Stopped:
		IF (GVL.PackTags.Command.CntrlCmd = ePMLCommand_Reset OR refMachine_control_cmd = MachineControlCommand.RESET OR GVL.fb_mcp.st_safety_door.button_reset) THEN
			fbMachine.eCommand	:= ePMLCommand_Reset;
		END_IF		
		IF (GVL.PackTags.Command.CntrlCmd = ePMLCommand_Start OR refMachine_control_cmd = MachineControlCommand.START)	
	 	AND (NOT (GVL.PackTags.Command.Parameter[1].Value <= 0) OR NOT (fbMachine.eMode = 1))
		AND stPMLUnitModeConfiguration[fbMachine.eMode].aStateDisabled[ePMLState_Idle] THEN
			fbMachine.eCommand	:= ePMLCommand_Start; 
		END_IF	
		IF refMachine_control_cmd = MachineControlCommand.STOP THEN
			refMachine_control_cmd	:= MachineControlCommand.DO_NOTHING;
		END_IF	
	ePMLState_Execute:	
		IF refMachine_control_cmd = MachineControlCommand.START THEN
			refMachine_control_cmd	:= MachineControlCommand.DO_NOTHING;
		END_IF
		IF GVL.PackTags.Command.CntrlCmd = ePMLCommand_Hold		
		AND( fbMachine.eMode =  1 OR fbMachine.eMode =  4 OR fbMachine.eMode = 2)  THEN
			fbMachine.eCommand	:= ePMLCommand_Hold;
		END_IF	
		IF GVL.PackTags.Command.CntrlCmd = ePMLCommand_Suspend	
		AND (fbMachine.eMode = 4 OR fbMachine.eMode = 1)THEN
			fbMachine.eCommand	:= ePMLCommand_Suspend;
		END_IF	 
	ePMLState_Held:	 
		IF GVL.PackTags.Command.CntrlCmd = ePMLCommand_Unhold THEN
			fbMachine.eCommand	:= ePMLCommand_Unhold;
		END_IF
	ePMLState_Suspended:
		IF GVL.PackTags.Command.CntrlCmd = ePMLCommand_Unsuspend THEN
		 	fbMachine.eCommand	:= ePMLCommand_Unsuspend;
		END_IF
	
END_CASE

/////////////////////////////abort/////////////////////////////	
IF 	fbMachine.eState <> ePMLState_Aborted AND fbMachine.eState <> ePMLState_Clearing THEN	
	IF GVL.PackTags.Command.CntrlCmd = ePMLCommand_Abort OR M_CheckError() THEN
		fbMachine.eCommand	:= ePMLCommand_Abort;
		refMachine_control_cmd	:= MachineControlCommand.DO_NOTHING;
	END_IF
END_IF
/////////////////////////////stop/////////////////////////////					
IF (GVL.PackTags.Command.CntrlCmd = ePMLCommand_Stop OR refMachine_control_cmd = MachineControlCommand.STOP) THEN
	fbMachine.eCommand	:= ePMLCommand_Stop;
	//
END_IF


2:
;
END_CASE



//
//Set the Packtags
M_SetPackTags();

//set the errors and warnings in Packtags
M_SetPackTagsErrorWarning();

//Call Visu
M_CallVisu();
///////////////////initialize unitmode and set 
IF GVL.PackTags.Command.UnitMode=ePMLProtUnitMode_Invalid THEN
	GVL.PackTags.Command.UnitMode	:= ePMLProtUnitMode_Production;
	GVL.PackTags.Command.Parameter[1].Value := 1;
END_IF
//Call FB_Machine
fbMachine(eModeCommand:= GVL.PackTags.Command.UnitMode,  eMode => GVL.PackTags.Status.UnitModeCurrent, eState =>GVL.PackTags.Status.StateCurrent);


//
CASE topicCallbackTest OF
	E_Topics.SAMPLE_SUBSCRRIBE_1:
		ADSLOGSTR(msgCtrlMask:= ADSLOG_MSGTYPE_LOG,msgFmtStr:='start publich test 1',strArg:='');
		dataCallbackTest.Topic	:= SAMPLE_SUBSCRRIBE_1;
		GVL.PubSubService.Publish(topic:= E_Topics.SAMPLE_SUBSCRRIBE_1,data:= dataCallbackTest);
		topicCallbackTest	:= E_Topics.UNKNOWN;
	E_Topics.SAMPLE_SUBSCRRIBE_2:
		ADSLOGSTR(msgCtrlMask:= ADSLOG_MSGTYPE_LOG,msgFmtStr:='start publich test 2',strArg:='');
		dataCallbackTest.Topic	:= SAMPLE_SUBSCRRIBE_2;
		GVL.PubSubService.Publish(topic:= E_Topics.SAMPLE_SUBSCRRIBE_2,data:= dataCallbackTest);
		topicCallbackTest	:= E_Topics.UNKNOWN;	
	E_Topics.SAMPLE_SUBSCRRIBE_3:
		ADSLOGSTR(msgCtrlMask:= ADSLOG_MSGTYPE_LOG,msgFmtStr:='start publich test 3',strArg:='');
		dataCallbackTest.Topic	:= SAMPLE_SUBSCRRIBE_3;
		GVL.PubSubService.Publish(topic:= E_Topics.SAMPLE_SUBSCRRIBE_3,data:= dataCallbackTest);
		topicCallbackTest	:= E_Topics.UNKNOWN;	
END_CASE

ACTION A_UnitModeConfig:
UserModeCofig(
	eMode							:= ePMLUnitMode_Service, 
	bDisableClearing				:= TRUE, 
	bDisableStarting				:= FALSE, 
	bDisableSuspended				:= FALSE, 
	bDisableStopping				:= TRUE, 
	bDisableAborting				:= TRUE, 
	bDisableHolding					:= TRUE, 
	bDisableHeld					:= TRUE, 
	bDisableUnholding				:= TRUE, 
	bDisableSuspending				:= TRUE, 
	bDisableUnsuspending			:= TRUE, 
	bDisableResetting				:= TRUE, 
	bDisableIdle					:= FALSE, 
	bDisableCompleting				:= TRUE, 
	bDisableComplete				:= FALSE, 
	bEnableUnitModeChangeStopped	:= TRUE, 
	bEnableUnitModeChangeIdle		:= TRUE, 
	bEnableUnitModeChangeSuspended	:= FALSE, 
	bEnableUnitModeChangeExecute	:= FALSE, 
	bEnableUnitModeChangeAborted	:= TRUE, 
	bEnableUnitModeChangeHeld		:= FALSE, 
	bEnableUnitModeChangeComplete	:= TRUE, 
	bError							=> , 
	nErrorId						=> );
END_ACTION

METHOD M_CallVisu
VAR_INPUT
END_VAR
//Calling FB_Visu
fbVisu(

	aKeyPressed				:= GVL.aKeyPressed,
	aUnitInfo				:= GVL.aUnitInfo, 
	bInvalidEntry			=> ,
	aCaption				=> GVL.aCaption,
	eModeVisu				=> ,
	eStateVisu				=> ,
	sUnitName				=> ,
	iFrameVisible			=> );
END_METHOD

METHOD M_CheckError : BOOL
VAR_INPUT
END_VAR

VAR
	
	
END_VAR
M_CheckError	:= FALSE;
FOR i:=1 TO GlobalParameters.MaxAlarms DO
	IF GVL.PackTags.Admin.Alarm[i].Trigger THEN
		M_CheckError	:= TRUE;
	END_IF
END_FOR
RETURN;//remove this while safety and air is ready
rTrig_error[0]();
rTrig_error[1]();
IF GVL.PackTags.Status.StateCurrent<>E_PMLState.ePMLState_Resetting THEN
	FOR i:=0 TO 10 DO
		IF rTrig_error[i].Q THEN
			GVL.pml_adminAlarm.M_SetAlarm(stAdmin:=GVL.PackTags.Admin,stAlarm:=GVL.alarm);
		END_IF
	END_FOR
END_IF

IF application.air_pressure_subsystem.current_air_pressure_state=CurrentAirPressureState.ERROR THEN
	GVL.alarm.Message	:= 'Air pressure is low';
	rTrig_error[0].CLK	:= TRUE;
ELSE
	rTrig_error[0].CLK	:= FALSE;
END_IF
IF application.safety.xError THEN
	GVL.alarm.Message	:= 'Safety input trigger';
	rTrig_error[1].CLK	:= TRUE;
ELSE
	rTrig_error[1].CLK	:= FALSE;
END_IF


IF application.safety.xError OR application.air_pressure_subsystem.current_air_pressure_state=CurrentAirPressureState.ERROR THEN
	M_CheckError	:= TRUE;
END_IF
END_METHOD

METHOD M_SetPackTags
VAR_INPUT
END_VAR
VAR	
END_VAR
//***************************Writing Data into GVL.PackTags***************************

//Parameters for the production
GVL.PackTags.Command.Parameter[1].ID				:= 1;
GVL.PackTags.Command.Parameter[1].Name				:= 'Quantity';
GVL.PackTags.Command.Parameter[1].Unit				:= 'Tote';

//Countig produced totes, see FB_sample
GVL.PackTags.Admin.ProdProcessedCount[1].ID			:= 1;
GVL.PackTags.Admin.ProdProcessedCount[1].Name		:= 'ToteFinish_Sample';
GVL.PackTags.Admin.ProdProcessedCount[1].Unit		:= 'Tote';





//Write the actual state and mode into the GVL.PackTags
GVL.PackTags.Status.StateCurrent					:= fbMachine.eState;
GVL.PackTags.Status.UnitModeCurrent					:= fbMachine.eMode;
GVL.PackTags.Status.StateRequested					:= fbMachine.eCommand;
GVL.PackTags.Status.UnitModeRequested				:= fbMachine.eModeCommand;
GVL.PackTags.Status.StateChangeInProcess			:= GVL.PackTags.Status.StateCurrent <> GVL.PackTags.Status.StateRequested;
GVL.PackTags.Status.UnitModeChangeInProcess			:= GVL.PackTags.Status.UnitModeCurrent <> GVL.PackTags.Status.UnitModeRequested;

//Write actual time and date in GVL.PackTags
fbLocalSystemTime(sNetID:= '', bEnable := TRUE);
GVL.PackTags.Admin.PlcDateTime[0]	:= fbLocalSystemTime.systemTime.wYear;
GVL.PackTags.Admin.PlcDateTime[1]	:= fbLocalSystemTime.systemTime.wMonth;
GVL.PackTags.Admin.PlcDateTime[2]	:= fbLocalSystemTime.systemTime.wDay;
GVL.PackTags.Admin.PlcDateTime[3]	:= fbLocalSystemTime.systemTime.wHour;
GVL.PackTags.Admin.PlcDateTime[4]	:= fbLocalSystemTime.systemTime.wMinute;
GVL.PackTags.Admin.PlcDateTime[5]	:= fbLocalSystemTime.systemTime.wSecond;
GVL.PackTags.Admin.PlcDateTime[6]	:= fbLocalSystemTime.systemTime.wMilliseconds;


//Set the productcounter to 0, when the production command is completed
fbTrigger(CLK:= (fbMachine.eState = ePMLState_Complete));
IF fbTrigger.Q OR GVL.stChangeIntoProduction.bYesReset THEN
	GVL.PackTags.Admin.ProdProcessedCount[1].Count	:= 0;
	GVL.PackTags.Command.Parameter[1].Value			:= 0;
	GVL.nVisuProductCommand							:= 0;
END_IF
END_METHOD

METHOD M_SetPackTagsErrorWarning
VAR_INPUT
END_VAR
//====================Error and Warnig setting========================
//Warnings
GVL.PackTags.Admin.Warning[1].Message	:= 'Invalid Production Command, command Products must be higher than 0';
GVL.PackTags.Admin.Warning[1].ID 		:= 1;

GVL.PackTags.Admin.Warning[2].Message	:= 'Invalid Mode Command, please try anothereone';
GVL.PackTags.Admin.Warning[2].ID		:= 2;


//====================Error and Warnig handling========================
//warning for invalid production command
IF GVL.PackTags.Status.UnitModeCurrent = ePMLProtUnitMode_Production AND GVL.PackTags.Status.StateCurrent = ePMLState_Idle AND GVL.PackTags.Command.CntrlCmd = ePMLCommand_Start AND GVL.PackTags.Command.Parameter[1].Value <= 0 THEN
	GVL.PackTags.Admin.Warning[1].Trigger :=TRUE;
ELSE
	GVL.PackTags.Admin.Warning[1].Trigger :=FALSE;
END_IF

//warning for invalid mode command
IF fbMachine.bInvalidModeCommandOut THEN
	GVL.PackTags.Admin.Warning[2].Trigger :=TRUE;
ELSE 
	GVL.PackTags.Admin.Warning[2].Trigger :=FALSE;
END_IF
END_METHOD

END_PROGRAM

// ---- Mian/FB_Machine.TcPOU
FUNCTION_BLOCK FB_Machine EXTENDS FB_Generic
VAR_INPUT

END_VAR
VAR_OUTPUT

END_VAR
VAR	

	
	stSubModuleInfo		: ARRAY [1..iSubModule] OF ST_PMLSubUnitInfo;	//Informations about the Subunits


	
	
END_VAR
VAR CONSTANT
	iSubModule	: UDINT :=1;
END_VAR

GVL.fb_sample(
	eModeCommand:= eModeCommand, 
	eCommand:= eCommand, 
	eMode=> , 
	eState=> stSubModuleInfo[iSubModule].eState, 
	bUndefinedDone=> , 
	bInvalidModeCommandOut=> , 
	bChangeIntoProduction=> );
stSubModuleInfo[iSubModule].Active		:= TRUE;

IF  GVL.fb_sample.bUndefinedDone  THEN
	bUndefinedDone := TRUE;
END_IF

//The fbStateMachine from FB_Machine gets the Information about the states and activity from the subunits
fbStateMachine.stSubUnitInfoRef.ArraySize		:= SIZEOF(stSubModuleInfo);
fbStateMachine.stSubUnitInfoRef.NoOfSubUnits	:= iSubModule;
fbStateMachine.stSubUnitInfoRef.pArray			:= ADR(stSubModuleInfo);



//Set unit information 
M_SetUnitInfo();


SUPER^();

{attribute 'object_name' := 'M_Clearing'}
METHOD M_Clearing

CASE fbUnitModeManager.eModeStatus OF
	ePMLProtUnitMode_Production:		//Production, Mantainance, Manual
		FOR i:=1 TO MaxAlarms DO
			GVL.pml_adminAlarm.M_AcknowledgeAlarm(stAdmin:=GVL.PackTags.Admin,stAlarm:=GVL.PackTags.Admin.Alarm[i]);
			GVL.pml_adminAlarm.M_ClearAlarm(stAdmin:=GVL.PackTags.Admin,stAlarm:=GVL.PackTags.Admin.Alarm[i]);
		END_FOR			
		IF MAIN.application.safety.M_reset() THEN
			IF MAIN.application.safety.xError THEN
				eCommand	:= ePMLCommand_Abort;
			ELSE
				M_StateComplete();
			END_IF
		END_IF	
		
	
	ePMLProtUnitMode_Maintenance, ePMLProtUnitMode_Manual, ePMLUnitMode_Service:
		M_StateComplete();
END_CASE
END_METHOD

{attribute 'object_name' := 'M_Resetting'}
METHOD M_Resetting
CASE fbUnitModeManager.eModeStatus OF
	ePMLProtUnitMode_Production:		//Production, Mantainance, Manual	
		IF MAIN.application.safety.M_reset() THEN
			IF MAIN.application.safety.xError THEN
				eCommand	:= ePMLCommand_Abort;
			ELSE
				M_StateComplete();
			END_IF
		END_IF	
		
	
	ePMLProtUnitMode_Maintenance, ePMLProtUnitMode_Manual, ePMLUnitMode_Service:
		M_StateComplete();
END_CASE
END_METHOD

METHOD M_SetUnitInfo
VAR_INPUT
END_VAR
GVL.aUnitInfo[eMachine].Name			:= 'fbMachine';
GVL.aUnitInfo[eMachine].ActMode			:= eMode;
GVL.aUnitInfo[eMachine].ActState		:= eState;

GVL.aUnitInfo[eSample].Name				:= 'fb_sample';
GVL.aUnitInfo[eSample].ActMode			:= GVL.fb_sample.eMode;
GVL.aUnitInfo[eSample].ActState			:= GVL.fb_sample.eState;
END_METHOD

{attribute 'object_name' := 'M_Starting'}
METHOD M_Starting
CASE fbUnitModeManager.eModeStatus OF
	ePMLProtUnitMode_Production:		//Production, Mantainance, Manual
		//Resetting all Commands and Value
		G_HMI.bAging_test	:= FALSE;
		M_StateComplete();
	ePMLProtUnitMode_Maintenance, ePMLProtUnitMode_Manual, ePMLUnitMode_Service:
		M_StateComplete();
END_CASE
END_METHOD

END_FUNCTION_BLOCK

// ---- Mian/FB_Visu.TcPOU
FUNCTION_BLOCK FB_Visu
VAR_INPUT
	
	// =============== Keys =====================================
	aKeyPressed						: ARRAY [1..12] OF BOOL;
	aUnitInfo						: ARRAY [1..12] OF ST_UnitInfo;
	aUnitCommand					: ARRAY [1..12] OF E_PMLCommand;
END_VAR
VAR_OUTPUT
	
	//=============== Cheking Button and entries =======================
	bInvalidEntry					: BOOL;						//Invalid entry, to produce products

	// =============== Keys =====================================
	aCaption						: ARRAY [1..12] OF STRING;	

	eModeVisu						: DINT;						// Mode for the 	StateChart	
	eStateVisu						: E_PMLState;				// State for the StateChart
	sUnitName						: STRING;
	iFrameVisible					: DINT;
	eUnitCommand					: E_PMLCommand;
END_VAR
VAR
	i								: DINT;

	// =============== Statechart variables ===================
	eUnitRepresentOnVisu			: E_UnitName := eMachine;	// Unit represent on Visu
		
	// =============== Warnings ===============================================
	sWarningVisu					: STRING;					// Descripton, name of the warning
	fbTimerWarning					: TON;						// Timer for visu textbox
	nWarningState					: INT :=0;					// State for representing warnings
	nWarningCount					: INT :=1;					// Variable to runs step by step trough the warningarray
	
	// =============== Errors ===============================================
	sAlarmVisu						: STRING;					// Descripton, name of the error
	fbTimerAlarm					: TON;						// Timer for visu textbox
	nAlarmState						: INT :=0;					// State for representing errors
	nAlarmCount						: INT :=1;					// Variable to runs step by step trough the errorarray
	
	nState							: INT;
	
END_VAR
VAR CONSTANT	
END_VAR

// =========================================================
// Select visible frame
aCaption[1] := 'Overview';
aCaption[2] := 'Machine';
aCaption[3] := 'Sample';


FOR i := 1 TO 11 DO
	IF aKeyPressed[i] THEN
		iFrameVisible := i - 1;		
	END_IF
END_FOR

IF iFrameVisible <= 1 THEN
	eModeVisu := aUnitInfo[1].ActMode;
	eStateVisu := aUnitInfo[1].ActState;
	sUnitName := aUnitInfo[1].Name;
	eUnitCommand	:= aUnitCommand[1];
ELSE
	eModeVisu := aUnitInfo[iFrameVisible].ActMode;
	eStateVisu := aUnitInfo[iFrameVisible].ActState;
	sUnitName := aUnitInfo[iFrameVisible].Name;
	aUnitCommand[iFrameVisible]	:= eUnitCommand;
END_IF

// =========================================================
// Visuazation functions
	
	// Checking production command
	M_ProductCommand();
	
	// Show Erorrs in Textbox
	M_Error_Warnings();

METHOD M_Error_Warnings
VAR_INPUT
END_VAR
//Show the Warnings on Visu
CASE nWarningState OF
	0:
		sWarningVisu					:= '';
		IF GVL.PackTags.Admin.Warning[nWarningCount].Trigger THEN
			fbTimerWarning.IN 		:= TRUE;
			fbTimerWarning.PT		:= T#3S;
			nWarningState			:= 1;
		ELSIF nWarningCount < 10 THEN
			nWarningCount		:= nWarningCount +1;
		ELSIF nWarningCount >= 10 THEN
			nWarningCount		:= 1;
		END_IF
	1:
		sWarningVisu 	:= GVL.PackTags.Admin.Warning[nWarningCount].Message;
		IF fbTimerWarning.Q THEN
			fbTimerWarning.IN 		:= FALSE;
			nWarningState			:= 0;
			
			IF nWarningCount < 10 THEN
				nWarningCount		:= nWarningCount +1;
			ELSIF nWarningCount >= 10 THEN
				nWarningCount		:= 1;
			END_IF
		END_IF
		
END_CASE	
fbTimerWarning();

//Show the Errors on Visu
CASE nAlarmState OF
	0:
		sAlarmVisu					:= '';
		IF GVL.PackTags.Admin.Alarm[nAlarmCount].Trigger THEN
			fbTimerAlarm.IN 		:= TRUE;
			fbTimerAlarm.PT		:= T#3S;
			nAlarmState			:= 1;
		ELSIF nAlarmCount < 10 THEN
			nAlarmCount		:= nAlarmCount +1;
		ELSIF nAlarmCount >= 10 THEN
			nAlarmCount		:= 1;
		END_IF
	1:
		sAlarmVisu 	:= GVL.PackTags.Admin.Alarm[nAlarmCount].Message;
		IF fbTimerAlarm.Q THEN
			fbTimerAlarm.IN 		:= FALSE;
			nAlarmState			:= 0;
			
			IF nAlarmCount < 10 THEN
				nAlarmCount		:= nAlarmCount +1;
			ELSIF nAlarmCount >= 10 THEN
				nAlarmCount		:= 1;
			END_IF
		END_IF
END_CASE
fbTimerAlarm();
END_METHOD

METHOD M_ProductCommand
//checking if productcommand is valid
IF	GVL.nVisuProductCommand > GVL.PackTags.Admin.ProdProcessedCount[1].Count	AND 
	GVL.nVisuProductCommand > GVL.PackTags.Admin.ProdProcessedCount[2].Count	AND 
	GVL.nVisuProductCommand > 0											THEN
			bInvalidEntry						:= FALSE;
			GVL.PackTags.Command.Parameter[1].Value := DINT_TO_REAL(GVL.nVisuProductCommand);
ELSIF	GVL.nVisuProductCommand < GVL.PackTags.Admin.ProdProcessedCount[1].Count	OR
		GVL.nVisuProductCommand < GVL.PackTags.Admin.ProdProcessedCount[2].Count	OR
		GVL.nVisuProductCommand < 0											THEN
			bInvalidEntry						:= TRUE;
END_IF
END_METHOD

END_FUNCTION_BLOCK

// ---- Ads/FB_Tote_Subsystem.TcPOU
FUNCTION_BLOCK FB_Tote_Subsystem
VAR_INPUT
END_VAR
VAR_OUTPUT
END_VAR
VAR
	status	: MachineStatus := MachineStatus.STOPPED;	
	current_air_pressure	: REAL;	
	machine_control_cmd	: MachineControlCommand;

	ton1	: TON;

	ton_heart_beat	: TON;
	bReset_ads_heart_beat	: BOOL;
	bTest	:BOOL;
	
	machine_current_status	: E_PMLState;


END_VAR

M_mapping();

machine_current_status	:= GVL.PackTags.Status.StateCurrent;

CASE machine_current_status OF
	ePMLState_Aborted,ePMLState_Aborting:
		status	:= MachineStatus.ERROR;
	ePMLState_Stopping:	
		status	:= MachineStatus.STOPPING;
	ePMLState_Stopped:
		status	:= MachineStatus.STOPPED;
	ePMLState_Resetting:	
		status	:= MachineStatus.RESETTING;
	ePMLState_Idle:	
		status	:= MachineStatus.READY;		
	ePMLState_Execute:	
		status	:= MachineStatus.RUNNING;			
		
END_CASE




/////////////////////////test/////////////////
ton1(PT:=T#1S);
IF bTest THEN//test ads heart beat
	ads_heart_beat(i:=1);
	bTest	:= FALSE;
END_IF
//////////////////////////ads heart beat/////////////////
ton_heart_beat(IN:=NOT bReset_ads_heart_beat,PT:=T#3S);
IF bReset_ads_heart_beat THEN
	bReset_ads_heart_beat	:= FALSE;
END_IF

{attribute 'TcRpcEnable'}
METHOD ads_heart_beat : BOOL
VAR_INPUT
	i	: INT;
END_VAR
ads_heart_beat	:= FALSE; 
bReset_ads_heart_beat	:= TRUE;
ads_heart_beat	:= TRUE;
END_METHOD

METHOD M_mapping : BOOL
VAR_INPUT
END_VAR
END_METHOD

{attribute 'TcRpcEnable'}
METHOD machine_control_command : BOOL
VAR_INPUT
	Command	: MachineControlCommand;
END_VAR
machine_control_command	:= FALSE; 

machine_control_cmd	:= Command;

machine_control_command	:= TRUE;
END_METHOD

END_FUNCTION_BLOCK

// ---- GlobalTextList.TcGTLO
TEXTLIST GlobalTextList
  55 = ' command Products: %i'
  323 = '%.2f'
  206 = '%.2f mm'
  829 = '%.2f MPa'
  1131 = '%.2r'
  740 = '%.3f mm'
  201 = '%s'
  209 = '+'
  210 = '-'
  54 = 'A C C I D E N T'
  18 = 'Abort'
  33 = 'Aborted'
  34 = 'Aborting'
  602 = 'Acc'
  843 = 'Actual Position'
  830 = 'Admin'
  773 = 'Aging test'
  5 = 'Alarm'
  61 = 'Average MachSpeed: %5.2f Package/min'
  203 = 'Axis Error '
  299 = 'Axis_bagOpen_0'
  618 = 'Axis_bagOpen_1'
  211 = 'Axis_bagOpen_2'
  743 = 'Axis_bagOpen_3'
  324 = 'Axis_vacuun_0'
  786 = 'Axis_vacuun_1'
  179 = 'BagOpen'
  959 = 'Bag_)'
  1353 = 'Bag_0'
  1316 = 'Bag_1'
  1317 = 'Bag_closed'
  517 = 'Bag_opened'
  81 = 'BELT ESTOP'
  1803 = 'bLoad_up'
  808 = 'Breaker OFF'
  486 = 'Breaker ON'
  1159 = 'buffer'
  327 = 'BUFFER SAFETY'
  732 = 'Buffer Stopper'
  16 = 'Clear'
  32 = 'Clearing'
  17 = 'Command'
  38 = 'Complete'
  1085 = 'Completing'
  58 = 'CurrentMachSpeed:%5.2f Package/min'
  1975 = 'DateTime'
  349 = 'Dec'
  216 = 'deg/s'
  217 = 'deg/s²'
  50 = 'Detection\nof metal'
  180 = 'DIO'
  68 = 'Do you want to change tp production mode?'
  662 = 'DOG'
  1080 = 'Down'
  673 = 'error'
  23 = 'Execute'
  19 = 'Execute\nComplete'
  924 = 'Extend'
  614 = 'extended'
  59 = 'Finished Metalboxes: %i'
  60 = 'Finished Plasticboxes: %i'
  56 = 'Finished Products: %i '
  801 = 'Flood Light'
  25 = 'Held'
  12 = 'Hold'
  26 = 'Holding'
  841 = 'HOME'
  248 = 'HomeDone'
  902 = 'ID'
  21 = 'Idle'
  136 = 'inbound'
  44 = 'INIT'
  4 = 'Invalid'
  1037 = 'Lamp'
  473 = 'Lift_down'
  293 = 'Lift_iuo'
  316 = 'Lift_up'
  51 = 'Light\nsensor'
  319 = 'Load'
  416 = 'Load_up'
  580 = 'Log In'
  234 = 'Log Out'
  1496 = 'LogOut'
  6 = 'Mantainance'
  7 = 'Manual'
  708 = 'Message'
  361 = 'Method'
  52 = 'Move belt\n+'
  53 = 'Move to\nwork position'
  491 = 'Muanal'
  737 = 'name'
  3 = 'No'
  1516 = 'NO.'
  258 = 'NO. '
  1043 = 'None'
  711 = 'Operator'
  1029 = 'outbound_end'
  787 = 'Pause'
  706 = 'photo_sens[1]or_start'
  1450 = 'PML '
  598 = 'Position Setting'
  1051 = 'Production'
  57 = 'Reset the Visu'
  30 = 'Reseting'
  1925 = 'Sample'
  36 = 'SC'
  1012 = 'sensor[0]'
  1257 = 'sensor[1]'
  82 = 'sensor[2]'
  774 = 'sensor[3]'
  1262 = 'sensor[4]'
  1137 = 'sensor[5]'
  794 = 'sensor[6]'
  512 = 'sensor[7]'
  681 = 'sensor_start[0]'
  1006 = 'sensor_start[1]'
  62 = 'Seperated Boxes: %i'
  415 = 'Service'
  102 = 'sStepID'
  99 = 'Jerk'
  839 = 'JOG BW'
  840 = 'JOG FW'
  1374 = 'lift'
  795 = 'LIFT'
  178 = 'Lift'
  926 = 'LIFT ESTOP'
  519 = 'LIFT STATION DETECTION'
  495 = 'LIGHT CURTAIN LEFT'
  39 = 'LIGHT CURTAIN RIGHT'
  413 = 'LOAD'
  897 = 'LOADING SAFETY'
  351 = 'Main'
  386 = 'MCP ESTOP'
  215 = 'mm/s'
  214 = 'mm/s²'
  207 = 'MOVE ABS'
  569 = 'Move relative'
  205 = 'Neg LS'
  677 = 'outbound'
  842 = 'photosensor[0]'
  79 = 'photosensor[1]'
  70 = 'photo_sensor[0]'
  919 = 'photo_sensor[1]'
  800 = 'photo_sensor_mute'
  925 = 'photo_sensor_mute_l'
  891 = 'photo_sensor_start'
  1003 = 'place'
  204 = 'Pos LS'
  844 = 'Power \nOn'
  359 = 'Power On'
  342 = 'ReM'
  1185 = 'ReM3'
  904 = 'ReM4'
  274 = 'ReM5'
  199 = 'Reset'
  10 = 'RESET'
  1651 = 'retract'
  934 = 'retracted'
  71 = 'ROBOT EAS'
  312 = 'ROBOT EES'
  72 = 'roller'
  1437 = 'Roller In'
  189 = 'roller[0]'
  709 = 'roller[1]'
  633 = 'roller[2]'
  687 = 'roller[3]'
  522 = 'roller_x'
  792 = 'roller_y'
  845 = 'RUN'
  634 = 'SAFETY DOOR'
  202 = 'SAFETY INPUT'
  617 = 'SAFETY OUTPUT'
  641 = 'sComponentID'
  438 = 'sComponent_ID'
  358 = 'sComponent_name'
  874 = 'sensor_mute'
  143 = 'sensor_mute_left'
  487 = 'sensor_mute_right'
  622 = 'Set absolute\nencoder as linear'
  454 = 'Set absolute\nencoder as rotation'
  208 = 'Set Point'
  14 = 'Set Pos to 0'
  332 = 'sEventType'
  714 = 'sEvent_MSG'
  245 = 'sID'
  220 = 'sMethod'
  1077 = 'Start'
  22 = 'Starting'
  67 = 'State Model\n%s'
  1034 = 'StepID'
  986 = 'sTime'
  198 = 'Stop'
  996 = 'STOP'
  31 = 'Stopped'
  35 = 'Stopping'
  1097 = 'Suspend'
  28 = 'Suspended'
  29 = 'Suspending'
  666 = 'Time'
  784 = 'tote_detection'
  585 = 'Type'
  13 = 'Unhold'
  24 = 'Unholding'
  20 = 'Unit Mode'
  780 = 'UNLOAD'
  809 = 'Unload'
  37 = 'Unsuspend'
  27 = 'Unsuspending'
  15 = 'Unuspend'
  407 = 'UP'
  505 = 'Up'
  848 = 'User'
  8 = 'UserMode 1'
  863 = 'valve_clamp[0]'
  396 = 'valve_lift'
  464 = 'valve_lift[0]'
  227 = 'valve_stopper'
  200 = 'Velocity'
  193 = 'WORKING SAFETY'
  1 = 'Yes'
  2 = 'Yes, with Reset'
END_TEXTLIST

// ---- VISUs/Templates/VIS_TemplateCommand.TcVIS
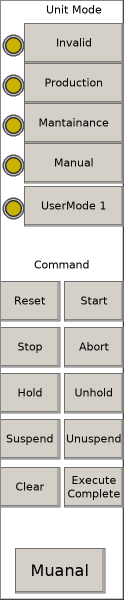
VISUALIZATION VIS_TemplateCommand  // 124x600
VAR_IN_OUT
	eModeCommand	: DINT;
	eStateCommand	: DINT;
	eModeStatus		: DINT;
	eStateStatus	: DINT;
	bModeChangeReq	: BOOL;
END_VAR
    Rectangle (0,0 124x600)
    Lamp1 (1,33 25x25), variable: (eModeStatus = 0), style: Lamp-Lamp1-Yellow
    Button (24,23 100x40), "Invalid", colour toggle: (eModeStatus = 0)
        tap bModeChangeReq
        OnMouseClick: execute { eModeCommand := 0; }
    Lamp1 (1,73 25x25), variable: (eModeStatus = 1), style: Lamp-Lamp1-Yellow
    Button (24,63 100x40), "Production"
        tap bModeChangeReq
        OnMouseClick: execute { eModeCommand := 1; }
    Lamp1 (1,113 25x25), variable: (eModeStatus = 2), style: Lamp-Lamp1-Yellow
    Button (24,103 100x40), "Mantainance"
        tap bModeChangeReq
        OnMouseClick: execute { eModeCommand := 2; }
    Lamp1 (1,153 25x25), variable: (eModeStatus = 3), style: Lamp-Lamp1-Yellow
    Button (24,143 100x40), "Manual"
        tap bModeChangeReq
        OnMouseClick: execute { eModeCommand := 3; }
    Lamp1 (1,196 25x25), variable: (eModeStatus = 4), style: Lamp-Lamp1-Yellow
    Button (24,186 100x40), "UserMode 1"
        tap bModeChangeReq
        OnMouseClick: execute { eModeCommand := 4; }
    Button (0,281 60x40), "Reset"
        OnMouseClick: execute { eStateCommand := 1; }
    Button (64,281 60x40), "Start"
        OnMouseClick: execute { eStateCommand := 2; }
    Button (0,327 60x40), "Stop"
        OnMouseClick: execute { eStateCommand := 3; }
    Button (0,373 60x40), "Hold"
        OnMouseClick: execute { eStateCommand := 4; }
    Button (64,373 60x40), "Unhold"
        OnMouseClick: execute { eStateCommand := 5; }
    Button (0,419 60x40), "Suspend"
        OnMouseClick: execute { eStateCommand := 6; }
    Button (64,419 60x40), "Unuspend"
        OnMouseClick: execute { eStateCommand := 7; }
    Button (0,467 60x40), "Clear"
        OnMouseClick: execute { eStateCommand := 9; }
    Label (0,255 124x20), "Command"
    Button (64,327 60x40), "Abort"
        OnMouseClick: execute { eStateCommand := 8; }
    Button (64,467 60x40), "Execute Complete"
        OnMouseClick: execute { MAIN.bExecuteComplete := TRUE; }
    Label (24,0 100x20), "Unit Mode"
    Button (15,548 90x45), "Muanal"
        p573394764: 16#FF00FF00
        OnMouseDown: execute {
            IF G_HMI.iPML_mainFrame	= 0 THEN
            	G_HMI.iPML_mainFrame	:= 1;
            ELSE
            	G_HMI.iPML_mainFrame	:= 0;
            END_IF
        }
END_VISUALIZATION

// ---- VISUs/Templates/VIS_TemplateKeys.TcVIS
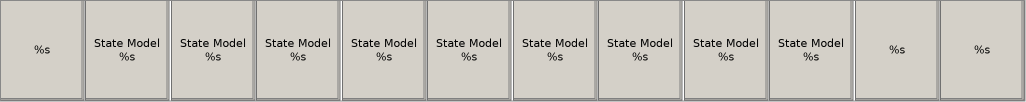
VISUALIZATION VIS_TemplateKeys  // 1026x102
VAR_INPUT
	Caption		: ARRAY [1..12] OF STRING;
END_VAR
VAR_IN_OUT
	KeyPressed	: ARRAY [1..12] OF BOOL;
END_VAR
    Button (0,0 84x100), "%s", text variable: Caption[1]
        tap KeyPressed[1]
    Button (85,0 84x100), "State Model %s", text variable: Caption[2]
        tap KeyPressed[2]
    Button (171,0 84x100), "State Model %s", text variable: Caption[3]
        tap KeyPressed[3]
    Button (256,0 84x100), "State Model %s", text variable: Caption[4]
        tap KeyPressed[4]
    Button (342,0 84x100), "State Model %s", text variable: Caption[5]
        tap KeyPressed[5]
    Button (427,0 84x100), "State Model %s", text variable: Caption[6]
        tap KeyPressed[6]
    Button (513,0 84x100), "State Model %s", text variable: Caption[7]
        tap KeyPressed[7]
    Button (598,0 84x100), "State Model %s", text variable: Caption[8]
        tap KeyPressed[8]
    Button (684,0 84x100), "State Model %s", text variable: Caption[9]
        tap KeyPressed[9]
    Button (769,0 84x100), "State Model %s", text variable: Caption[10]
        tap KeyPressed[10]
    Button (855,0 84x100), "%s", text variable: Caption[11]
        tap KeyPressed[11]
    Button (940,0 84x100), "%s", text variable: Caption[12]
        tap KeyPressed[12]
END_VISUALIZATION

// ---- VISUs/Templates/VIS_TemplateMachine.TcVIS
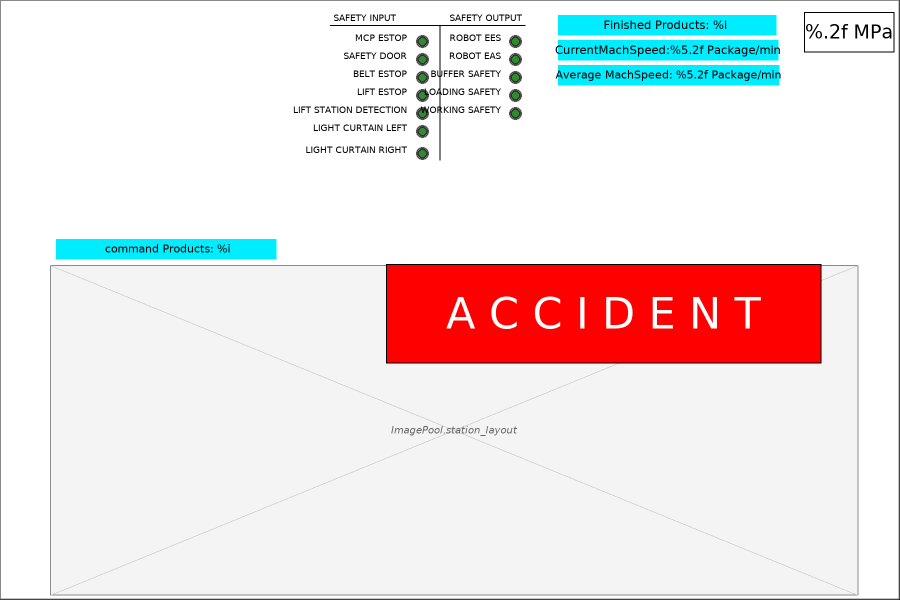
VISUALIZATION VIS_TemplateMachine  // 900x600
    Rectangle (0,0 900x600)
    Image (50,265 808x330), image: ImagePool.station_layout
    Rectangle (386,264 435x99), "A C C I D E N T", invisible if: NOT (MAIN.application.tote_subsystem.status=MachineStatus.ERROR)
    Rectangle (56,239 220x20), "command Products: %i", text variable: GVL.PackTags.Command.Parameter[1].Value, colour toggle: (MAIN.fbVisu.bInValidEntry OR GVL.PackTags.Admin.Warning[1].Trigger), invisible if: NOT ( MAIN.fbMachine.eMode = 1)
        OnMouseClick: write GVL.nVisuProductCommand via Default
    Rectangle (558,15 218x20), "Finished Products: %i", text variable: GVL.PackTags.Admin.ProdProcessedCount[1].Count, invisible if: NOT ( MAIN.fbMachine.eMode = 1)
    Rectangle (558,40 220x20), "CurrentMachSpeed:%5.2f Package/min", text variable: GVL.PackTags.Status.CurMachineSpeed, invisible if: NOT ( MAIN.fbMachine.eMode = 1)
    Rectangle (558,65 221x20), "Average MachSpeed: %5.2f Package/min", text variable: GVL.PackTags.Status.MachineSpeed, invisible if: NOT ( MAIN.fbMachine.eMode = 1)
    Lamp1 (415,34 15x15), variable: MAIN.application.safety.mcp_estop, style: Lamp-Lamp1-Green
    Label (330,34 80x8), "MCP ESTOP"
    Lamp1 (415,70 15x15), variable: MAIN.application.safety.belt_estop, style: Lamp-Lamp1-Green
    Label (330,70 80x8), "BELT ESTOP"
    Lamp1 (415,88 15x15), variable: MAIN.application.safety.lift_estop, style: Lamp-Lamp1-Green
    Label (330,88 80x8), "LIFT ESTOP"
    Lamp1 (415,106 15x15), variable: MAIN.application.safety.lift_station_detection, style: Lamp-Lamp1-Green
    Label (330,106 80x8), "LIFT STATION DETECTION"
    Lamp1 (415,52 15x15), variable: MAIN.application.safety.mcp_safetyDoor, style: Lamp-Lamp1-Green
    Label (330,52 80x8), "SAFETY DOOR"
    Lamp1 (415,124 15x15), variable: MAIN.application.safety.lift_lightCurtain_left, style: Lamp-Lamp1-Green
    Label (330,124 80x8), "LIGHT CURTAIN LEFT"
    Lamp1 (415,146 15x15), variable: MAIN.application.safety.lift_lightCurtain_right, style: Lamp-Lamp1-Green
    Label (330,146 80x8), "LIGHT CURTAIN RIGHT"
    Lamp1 (508,34 15x15), variable: MAIN.application.safety.robot_EES, style: Lamp-Lamp1-Green
    Label (444,34 60x8), "ROBOT EES"
    Lamp1 (508,70 15x15), variable: MAIN.application.safety.buffer_safety, style: Lamp-Lamp1-Green
    Label (444,70 60x8), "BUFFER SAFETY"
    Lamp1 (508,88 15x15), variable: MAIN.application.safety.loading_safety, style: Lamp-Lamp1-Green
    Label (444,88 60x8), "LOADING SAFETY"
    Lamp1 (508,106 15x15), variable: MAIN.application.safety.working_safety, style: Lamp-Lamp1-Green
    Label (444,106 60x8), "WORKING SAFETY"
    Lamp1 (508,52 15x15), variable: MAIN.application.safety.robot_EAS, style: Lamp-Lamp1-Green
    Label (444,52 60x8), "ROBOT EAS"
    Line (440,160) (440,25)
    Label (315,12 100x12), "SAFETY INPUT"
    Label (436,12 100x12), "SAFETY OUTPUT"
    Line (330,25) (525,25)
    Rectangle (804,12 90x40), "%.2f MPa", text variable: MAIN.application.air_pressure_subsystem.current_air_pressure
END_VISUALIZATION

// ---- VISUs/VISUs/Menu.TcVIS
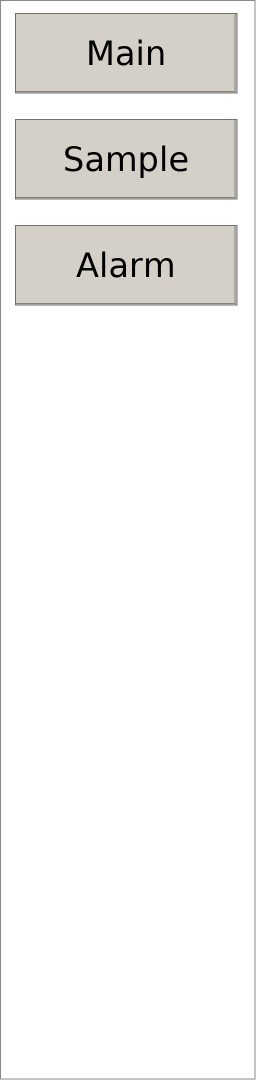
VISUALIZATION Menu  // 256x1080
    Button (15,119 222x80), "Sample", colour toggle: G_HMI.iMainFrame =1
        p573394764: 16#FF00FF00
        OnMouseDown: execute { G_HMI.iMainFrame	:= 1; }
    Button (15,225 222x80), "Alarm", colour toggle: G_HMI.iMainFrame =2
        p573394764: 16#FF00FF00
        OnMouseDown: execute { G_HMI.iMainFrame	:= 2; }
    Button (15,13 222x80), "Main", colour toggle: G_HMI.iMainFrame =0
        p573394764: 16#FF00FF00
        OnMouseDown: execute { G_HMI.iMainFrame	:= 0; }
END_VISUALIZATION

// ---- VISUs/VISUs/visu_manual.TcVIS
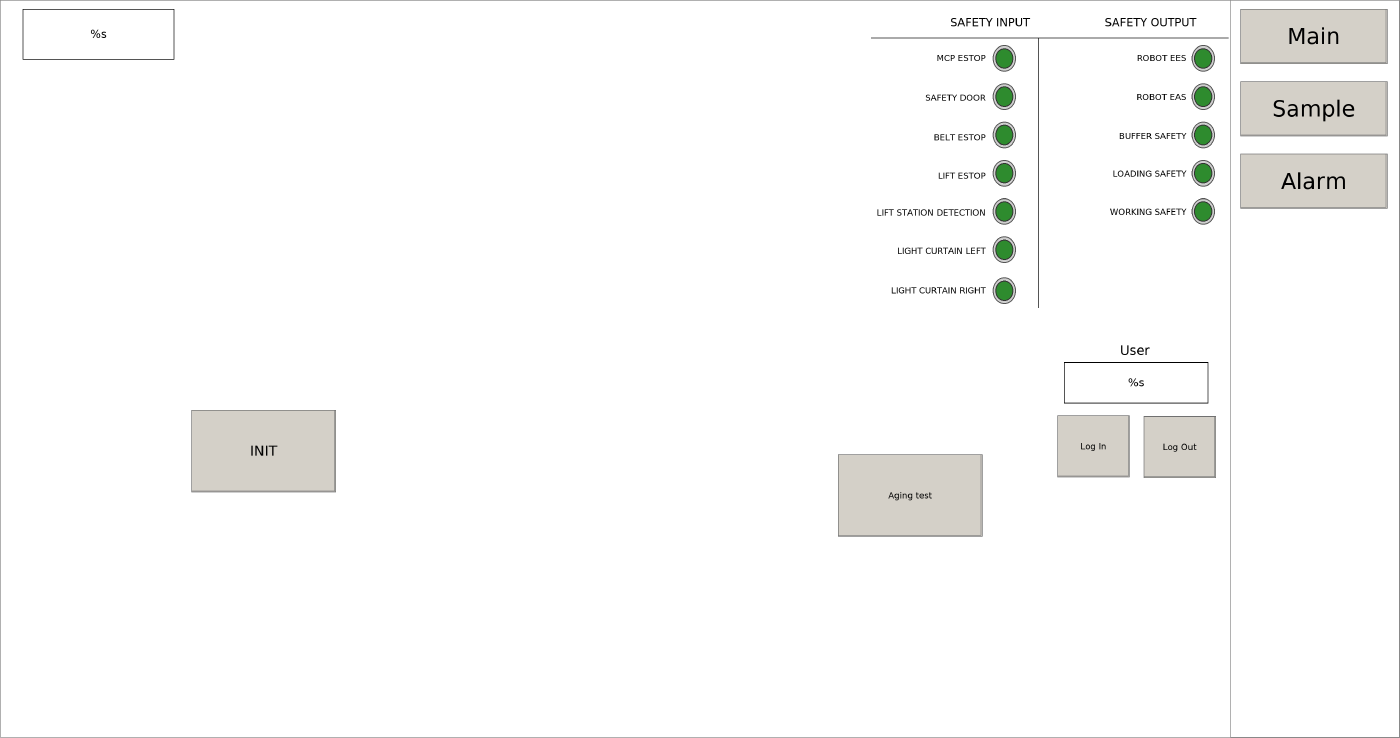
VISUALIZATION visu_manual  // 2048x1080
    Frame (0,0 1800x1080), frame switch variable: G_HMI.iMainFrame
        shows visu_operation()
        shows visu_sample()
        shows v_alarm()
        shows v_IO_fixtureClamp()
        shows visu_working()
        shows v_alarm()
    Frame (1800,0 248x1080), frame switch variable: G_HMI.iMainFrame
        shows Menu()
        shows visu_working()
        shows v_IO_fixtureClamp()
        shows visu_buffer()
        shows visu_loading()
        shows v_alarm()
END_VISUALIZATION

// ---- VISUs/VISUs/visu_operation.TcVIS
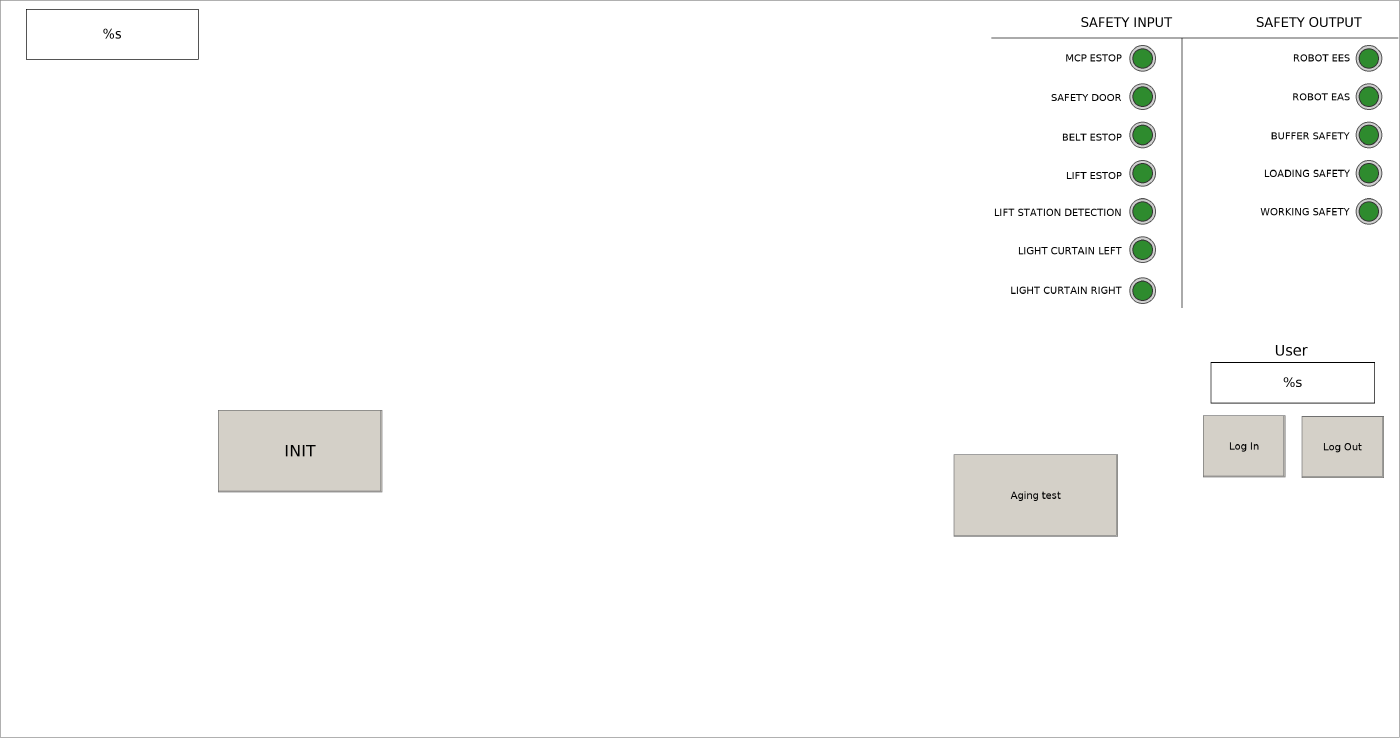
VISUALIZATION visu_operation  // 2048x1080
    Button (319,600 240x120), "INIT", colour toggle: G_HMI.bInit
        OnMouseDown: execute { G_HMI.bInit	:= TRUE; }
        OnMouseUp: execute { G_HMI.bInit	:= FALSE; }
    Lamp1 (1649,63 45x45), variable: MAIN.application.safety.mcp_estop, style: Lamp-Lamp1-Green
    Label (1344,70 300x30), "MCP ESTOP"
    Lamp1 (1649,175 45x45), variable: MAIN.application.safety.belt_estop, style: Lamp-Lamp1-Green
    Label (1344,186 300x30), "BELT ESTOP"
    Lamp1 (1649,231 45x45), variable: MAIN.application.safety.lift_estop, style: Lamp-Lamp1-Green
    Label (1344,244 300x26), "LIFT ESTOP"
    Lamp1 (1649,287 45x45), variable: MAIN.application.safety.lift_station_detection, style: Lamp-Lamp1-Green
    Label (1344,298 300x26), "LIFT STATION DETECTION"
    Lamp1 (1649,119 45x45), variable: MAIN.application.safety.mcp_safetyDoor, style: Lamp-Lamp1-Green
    Label (1344,128 300x30), "SAFETY DOOR"
    Lamp1 (1649,343 45x45), variable: MAIN.application.safety.lift_lightCurtain_left, style: Lamp-Lamp1-Green
    Label (1344,352 300x30), "LIGHT CURTAIN LEFT"
    Lamp1 (1649,403 45x45), variable: MAIN.application.safety.lift_lightCurtain_right, style: Lamp-Lamp1-Green
    Label (1344,410 300x30), "LIGHT CURTAIN RIGHT"
    Lamp1 (1980,63 45x45), variable: MAIN.application.safety.robot_EES, style: Lamp-Lamp1-Green
    Label (1728,70 250x30), "ROBOT EES"
    Lamp1 (1980,175 45x45), variable: MAIN.application.safety.buffer_safety, style: Lamp-Lamp1-Green
    Label (1728,184 250x30), "BUFFER SAFETY"
    Lamp1 (1980,231 45x45), variable: MAIN.application.safety.loading_safety, style: Lamp-Lamp1-Green
    Label (1728,241 250x26), "LOADING SAFETY"
    Lamp1 (1980,287 45x45), variable: MAIN.application.safety.working_safety, style: Lamp-Lamp1-Green
    Label (1728,297 250x26), "WORKING SAFETY"
    Lamp1 (1980,119 45x45), variable: MAIN.application.safety.robot_EAS, style: Lamp-Lamp1-Green
    Label (1728,127 250x30), "ROBOT EAS"
    Line (1729,450) (1729,55)
    Label (1523,18 250x30), "SAFETY INPUT"
    Label (1790,18 250x30), "SAFETY OUTPUT"
    Line (1450,55) (2045,55)
    Button (1395,665 240x120), "Aging test", colour toggle: G_HMI.bAging_test
        toggle G_HMI.bAging_test
    Rectangle (38,13 252x74), "%s"
    Rectangle (1771,530 240x60), "%s", text variable: G_HMI.sLoginnedUser
    Button (1904,609 120x90), "Log Out"
        OnMouseDown: VisuUserMgmt Type=Logout
    Button (1760,608 120x90), "Log In"
        OnMouseDown: VisuUserMgmt Type=Login
    Label (1814,498 150x30), "User"
END_VISUALIZATION

// ---- VISUs/VISUs/v_alarm.TcVIS
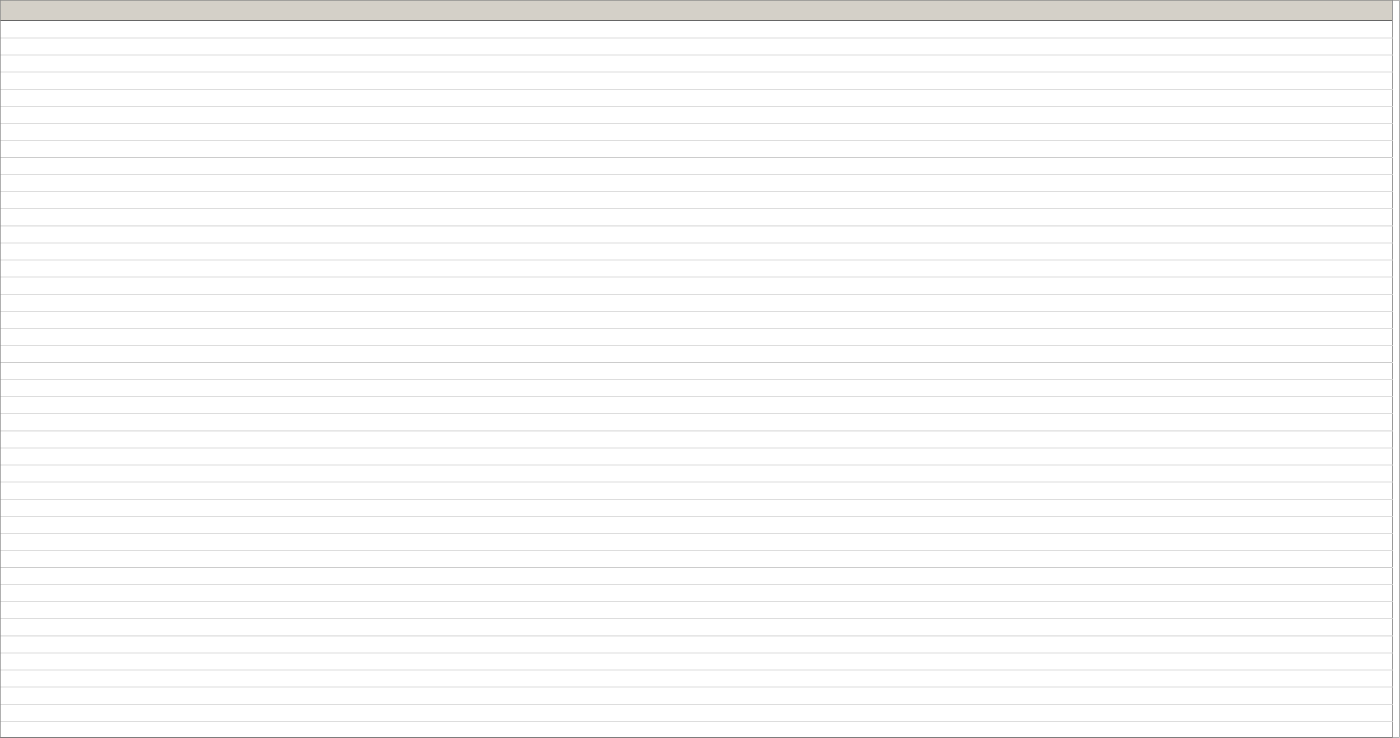
VISUALIZATION v_alarm  // 2048x1080
    Table (-11,0 2048x1080), data array: GVL.PackTags.Admin.Alarm
        p3104783080: GVL.fb_buffer.fb_rollers[INDEX].AxisRef
        p2501879983: GVL.fb_buffer.fb_rollers[INDEX].current_tote_status
        p7306298: GVL.fb_buffer.fb_rollers[INDEX].ton_timeout
        p1933151965: GVL.fb_buffer.fb_rollers[INDEX].eStates
        p3863566920: GVL.fb_buffer.fb_rollers[INDEX].iStateTemp
        p2192122294: GVL.fb_buffer.fb_rollers[INDEX].errorMessage
        p400160035: GVL.fb_buffer.fb_rollers[INDEX].xError
        p1265227338: GVL.fb_buffer.fb_rollers[INDEX].rPos_up
        p3726181087: GVL.fb_buffer.fb_rollers[INDEX].rPos_down
        p3854506369: GVL.PackTags.Admin.Alarm[INDEX].Trigger
        p1892666644: GVL.PackTags.Admin.Alarm[INDEX].ID
        p338671338: GVL.PackTags.Admin.Alarm[INDEX].Value
        p2170511999: GVL.PackTags.Admin.Alarm[INDEX].Message
        p3723444502: GVL.PackTags.Admin.Alarm[INDEX].Category
        p1218418051: GVL.PackTags.Admin.Alarm[INDEX].DateTime
        p746581629: GVL.PackTags.Admin.Alarm[INDEX].AckDateTime
END_VISUALIZATION

// ---- VISUs/visu_main.TcVIS
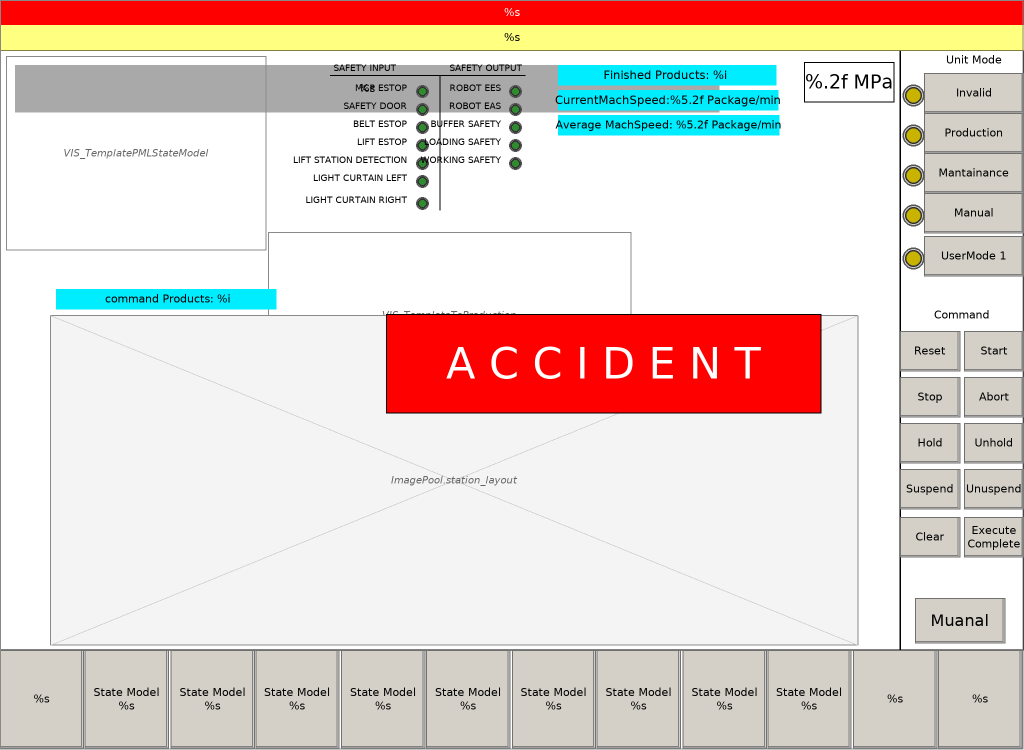
VISUALIZATION visu_main  // 1024x750
    Frame (0,50 900x600), invisible if: MAIN.fbVisu.iFrameVisible = 0 OR MAIN.fbMachine.bChangeIntoProduction
        shows VIS_TemplatePMLStateModel(ePMLUnitMode := MAIN.fbVisu.eModeVisu, ePMLState := MAIN.fbVisu.eStateVisu, eStateCommand := MAIN.fbVisu.eUnitCommand)
        shows VIS_TemplatePMLStateModel()
    Frame (268,232 363x166), invisible if: NOT MAIN.fbMachine.bChangeIntoProduction
        shows VIS_TemplateToProduction(stChangeIntoProduction := GVL.stChangeIntoProduction)
    Textfield (15,65 704x47), "%s", text variable: MAIN.fbVisu.sUnitName, invisible if: MAIN.fbVisu.iFrameVisible = 0 OR MAIN.fbMachine.bChangeIntoProduction
    Frame (0,50 900x600), invisible if: MAIN.fbVisu.iFrameVisible > 0 OR MAIN.fbMachine.bChangeIntoProduction, frame switch variable: G_HMI.iPML_mainFrame
        shows VIS_TemplateMachine()
        shows visu_manual()
    Rectangle (0,0 1024x25), "%s", text variable: MAIN.fbVisu.sAlarmVisu, invisible if: (MAIN.fbMachine.bChangeIntoProduction OR MAIN.fbVisu.sAlarmVisu = '')
    Frame (900,50 124x600)
        shows VIS_TemplateCommand(eModeCommand := GVL.PackTags.Command.UnitMode, eStateCommand := GVL.PackTags.Command.CntrlCmd, eModeStatus := GVL.PackTags.Status.UnitModeCurrent, eStateStatus := GVL.PackTags.Status.StateCurrent, bModeChangeReq := GVL.PackTags.Command.UnitModeChangeRequest)
    Frame (0,650 1024x100)
        shows VIS_TemplateKeys(Caption := GVL.aCaption, KeyPressed := GVL.aKeyPressed)
    Frame (6,56 260x194), invisible if: MAIN.fbVisu.iFrameVisible > 0 OR MAIN.fbMachine.bChangeIntoProduction OR G_HMI.iPML_mainFrame=1
        shows VIS_TemplatePMLStateModel(ePMLUnitMode := GVL.PackTags.Status.UnitModeCurrent, ePMLState := GVL.PackTags.Status.StateCurrent, eStateCommand := MAIN.fbMachine.eCommand)
    Rectangle (0,25 1024x25), "%s", text variable: MAIN.fbVisu.sWarningVisu, invisible if: (MAIN.fbMachine.bChangeIntoProduction OR MAIN.fbVisu.sWarningVisu ='')
END_VISUALIZATION
